  MoveL 5258 to (-75.49, 1.51, -146.03) mm, rotated rx -9.61 ry -16.54 rz -54.03 deg; joints [-10.747, -61.627, 111.301, 199.132, 34.736, -117.948, -415]
  MoveL 5259 to (-75.17, 1.21, -145.97) mm, rotated rx -9.61 ry -16.54 rz -54.03 deg; joints [-10.746, -61.652, 111.337, 199.128, 34.747, -117.942, -415]
  MoveL 5260 to (-74.81, 0.9, -145.93) mm, rotated rx -9.61 ry -16.54 rz -54.03 deg; joints [-10.747, -61.679, 111.378, 199.12, 34.76, -117.933, -415]
  MoveL 5261 to (-74.43, 0.59, -145.92) mm, rotated rx -9.61 ry -16.54 rz -54.03 deg; joints [-10.748, -61.706, 111.42, 199.111, 34.774, -117.923, -415]
  MoveL 5262 to (-74.01, 0.26, -145.91) mm, rotated rx -9.61 ry -16.54 rz -54.03 deg; joints [-10.75, -61.734, 111.466, 199.099, 34.79, -117.911, -415]
  MoveL 5263 to (-73.59, -0.06, -145.91) mm, rotated rx -9.61 ry -16.54 rz -54.03 deg; joints [-10.753, -61.762, 111.51, 199.087, 34.805, -117.899, -415]
  MoveL 5264 to (-73.18, -0.36, -145.93) mm, rotated rx -9.61 ry -16.54 rz -54.03 deg; joints [-10.756, -61.788, 111.554, 199.075, 34.821, -117.886, -415]
  MoveL 5265 to (-72.78, -0.65, -145.94) mm, rotated rx -9.61 ry -16.54 rz -54.03 deg; joints [-10.758, -61.814, 111.596, 199.062, 34.836, -117.873, -415]
  MoveL 5266 to (-72.42, -0.94, -145.92) mm, rotated rx -9.61 ry -16.54 rz -54.03 deg; joints [-10.76, -61.839, 111.636, 199.054, 34.849, -117.864, -415]
  MoveL 5267 to (-72.07, -1.24, -145.88) mm, rotated rx -9.61 ry -16.54 rz -54.03 deg; joints [-10.76, -61.865, 111.675, 199.047, 34.862, -117.855, -415]
  MoveL 5268 to (-71.66, -1.6, -145.83) mm, rotated rx -9.61 ry -16.54 rz -54.03 deg; joints [-10.76, -61.895, 111.722, 199.039, 34.877, -117.846, -415]
  MoveL 5269 to (-71.13, -2.06, -145.77) mm, rotated rx -9.61 ry -16.54 rz -54.03 deg; joints [-10.761, -61.935, 111.781, 199.028, 34.896, -117.834, -415]
  MoveL 5270 to (-70.63, -2.48, -145.75) mm, rotated rx -9.61 ry -16.54 rz -54.03 deg; joints [-10.763, -61.97, 111.836, 199.016, 34.914, -117.821, -415]
  MoveL 5271 to (-68.56, -4.07, -145.75) mm, rotated rx -9.61 ry -16.54 rz -54.03 deg; joints [-10.775, -62.109, 112.059, 198.957, 34.991, -117.76, -415]
  MoveL 5272 to (-68.07, -4.47, -145.71) mm, rotated rx -9.61 ry -16.54 rz -54.03 deg; joints [-10.776, -62.143, 112.112, 198.946, 35.008, -117.748, -415]
  MoveL 5273 to (-67.65, -4.83, -145.65) mm, rotated rx -9.61 ry -16.54 rz -54.03 deg; joints [-10.776, -62.174, 112.159, 198.939, 35.024, -117.739, -415]
  MoveL 5274 to (-67.49, -4.97, -145.51) mm, rotated rx -9.61 ry -16.54 rz -54.03 deg; joints [-10.771, -62.187, 112.178, 198.944, 35.031, -117.741, -415]
  MoveL 5275 to (-67.59, -4.89, -145.24) mm, rotated rx -9.61 ry -16.54 rz -54.03 deg; joints [-10.76, -62.181, 112.17, 198.964, 35.031, -117.754, -415]
  MoveL 5276 to (-67.93, -4.58, -144.84) mm, rotated rx -9.61 ry -16.54 rz -54.03 deg; joints [-10.741, -62.158, 112.136, 198.999, 35.025, -117.78, -415]
  MoveL 5277 to (-68.27, -5.55, -144.03) mm, rotated rx -9.61 ry -16.54 rz -54.03 deg; joints [-10.709, -62.222, 112.153, 199.074, 34.987, -117.841, -415]
  MoveL 5278 to (-67.69, -7.45, -143.82) mm, rotated rx -9.61 ry -16.54 rz -54.03 deg; joints [-10.707, -62.359, 112.27, 199.087, 34.969, -117.855, -415]
  MoveL 5279 to (-67.08, -9.36, -143.66) mm, rotated rx -9.61 ry -16.54 rz -54.03 deg; joints [-10.707, -62.497, 112.39, 199.095, 34.951, -117.865, -415]
  MoveL 5280 to (-66.45, -11.32, -143.5) mm, rotated rx -9.61 ry -16.54 rz -54.03 deg; joints [-10.708, -62.639, 112.512, 199.103, 34.933, -117.875, -415]
  MoveL 5281 to (-65.89, -13.11, -143.21) mm, rotated rx -9.61 ry -16.54 rz -54.03 deg; joints [-10.702, -62.769, 112.625, 199.121, 34.917, -117.892, -415]
  MoveL 5282 to (-65.24, -15.12, -143.02) mm, rotated rx -9.61 ry -16.54 rz -54.03 deg; joints [-10.701, -62.915, 112.75, 199.131, 34.898, -117.904, -415]
  MoveL 5283 to (-64.56, -17.23, -142.84) mm, rotated rx -9.61 ry -16.54 rz -54.03 deg; joints [-10.701, -63.068, 112.882, 199.142, 34.877, -117.917, -415]
  MoveL 5284 to (-63.86, -19.36, -142.75) mm, rotated rx -9.61 ry -16.54 rz -54.03 deg; joints [-10.705, -63.223, 113.014, 199.145, 34.856, -117.925, -415]
  MoveL 5285 to (-63, -21.95, -142.66) mm, rotated rx -9.61 ry -16.54 rz -54.03 deg; joints [-10.711, -63.411, 113.175, 199.149, 34.829, -117.934, -415]
  MoveL 5286 to (-62.38, -23.8, -142.56) mm, rotated rx -9.61 ry -16.54 rz -54.03 deg; joints [-10.713, -63.546, 113.292, 199.153, 34.811, -117.942, -415]
  MoveL 5287 to (-61.8, -25.54, -142.34) mm, rotated rx -9.61 ry -16.54 rz -54.03 deg; joints [-10.711, -63.673, 113.401, 199.166, 34.795, -117.955, -415]
  MoveL 5288 to (-61.16, -27.45, -142.15) mm, rotated rx -9.61 ry -16.54 rz -54.03 deg; joints [-10.71, -63.813, 113.521, 199.177, 34.776, -117.968, -415]
  MoveL 5289 to (-60.47, -29.47, -142.03) mm, rotated rx -9.61 ry -16.54 rz -54.03 deg; joints [-10.712, -63.96, 113.647, 199.183, 34.755, -117.978, -415]
  MoveL 5290 to (-59.79, -31.47, -141.85) mm, rotated rx -9.61 ry -16.54 rz -54.03 deg; joints [-10.712, -64.106, 113.772, 199.193, 34.736, -117.99, -415]
  MoveL 5291 to (-59.11, -33.47, -141.73) mm, rotated rx -9.61 ry -16.54 rz -54.03 deg; joints [-10.715, -64.253, 113.897, 199.2, 34.715, -118, -415]
  MoveL 5292 to (-58.4, -35.53, -141.55) mm, rotated rx -9.61 ry -16.54 rz -54.03 deg; joints [-10.715, -64.404, 114.026, 199.21, 34.694, -118.012, -415]
  MoveL 5293 to (-57.7, -37.55, -141.43) mm, rotated rx -9.61 ry -16.54 rz -54.03 deg; joints [-10.717, -64.551, 114.152, 199.216, 34.673, -118.022, -415]
  MoveL 5294 to (-56.99, -39.56, -141.2) mm, rotated rx -9.61 ry -16.54 rz -54.03 deg; joints [-10.715, -64.7, 114.279, 199.23, 34.653, -118.036, -415]
  MoveL 5295 to (-56.29, -41.58, -141.09) mm, rotated rx -9.61 ry -16.54 rz -54.03 deg; joints [-10.718, -64.848, 114.405, 199.236, 34.631, -118.047, -415]
  MoveL 5296 to (-55.59, -43.59, -140.97) mm, rotated rx -9.61 ry -16.54 rz -54.03 deg; joints [-10.721, -64.996, 114.53, 199.242, 34.609, -118.057, -415]
  MoveL 5297 to (-54.86, -45.6, -140.75) mm, rotated rx -9.61 ry -16.54 rz -54.03 deg; joints [-10.719, -65.144, 114.657, 199.255, 34.59, -118.071, -415]
  MoveL 5298 to (-54.16, -47.41, -140.55) mm, rotated rx -9.61 ry -16.54 rz -54.03 deg; joints [-10.717, -65.279, 114.776, 199.265, 34.575, -118.082, -415]
  MoveL 5299 to (-53.46, -49.03, -140.26) mm, rotated rx -9.61 ry -16.54 rz -54.03 deg; joints [-10.712, -65.401, 114.888, 199.28, 34.567, -118.094, -415]
  MoveL 5300 to (-52.73, -50.49, -139.85) mm, rotated rx -9.61 ry -16.54 rz -54.03 deg; joints [-10.701, -65.514, 114.997, 199.299, 34.566, -118.107, -415]
  MoveL 5301 to (-52.69, -49, -138.92) mm, rotated rx -9.61 ry -16.54 rz -54.03 deg; joints [-10.658, -65.419, 114.96, 199.342, 34.629, -118.12, -415]
  MoveL 5302 to (-52.62, -49.58, -138.91) mm, rotated rx -9.61 ry -16.54 rz -54.03 deg; joints [-10.659, -65.459, 114.984, 199.347, 34.615, -118.128, -415]
  MoveL 5303 to (-52.59, -50.11, -138.89) mm, rotated rx -9.61 ry -16.54 rz -54.03 deg; joints [-10.66, -65.495, 115.005, 199.354, 34.599, -118.137, -415]
  MoveL 5304 to (-52.61, -50.58, -138.83) mm, rotated rx -9.61 ry -16.54 rz -54.03 deg; joints [-10.658, -65.527, 115.02, 199.365, 34.584, -118.148, -415]
  MoveL 5305 to (-52.65, -51.02, -138.76) mm, rotated rx -9.61 ry -16.54 rz -54.03 deg; joints [-10.656, -65.557, 115.032, 199.376, 34.568, -118.16, -415]
  MoveL 5306 to (-52.73, -51.48, -138.71) mm, rotated rx -9.61 ry -16.54 rz -54.03 deg; joints [-10.655, -65.587, 115.042, 199.388, 34.549, -118.174, -415]
  MoveL 5307 to (-52.83, -51.96, -138.68) mm, rotated rx -9.61 ry -16.54 rz -54.03 deg; joints [-10.654, -65.618, 115.05, 199.4, 34.527, -118.188, -415]
  MoveL 5308 to (-52.96, -52.47, -138.66) mm, rotated rx -9.61 ry -16.54 rz -54.03 deg; joints [-10.654, -65.65, 115.057, 199.412, 34.503, -118.203, -415]
  MoveL 5309 to (-53.1, -52.97, -138.66) mm, rotated rx -9.61 ry -16.54 rz -54.03 deg; joints [-10.655, -65.682, 115.063, 199.424, 34.479, -118.217, -415]
  MoveL 5310 to (-53.21, -53.43, -138.65) mm, rotated rx -9.61 ry -16.54 rz -54.03 deg; joints [-10.655, -65.711, 115.07, 199.435, 34.458, -118.23, -415]
  MoveL 5311 to (-53.3, -53.84, -138.63) mm, rotated rx -9.61 ry -16.54 rz -54.03 deg; joints [-10.655, -65.738, 115.077, 199.445, 34.439, -118.242, -415]
  MoveL 5312 to (-53.41, -54.31, -138.61) mm, rotated rx -9.61 ry -16.54 rz -54.03 deg; joints [-10.655, -65.768, 115.083, 199.456, 34.417, -118.256, -415]
  MoveL 5313 to (-53.55, -54.82, -138.61) mm, rotated rx -9.61 ry -16.54 rz -54.03 deg; joints [-10.656, -65.8, 115.089, 199.467, 34.393, -118.27, -415]
  MoveL 5314 to (-53.7, -55.41, -138.59) mm, rotated rx -9.61 ry -16.54 rz -54.03 deg; joints [-10.656, -65.838, 115.097, 199.482, 34.365, -118.288, -415]
  MoveL 5315 to (-53.86, -56.09, -138.55) mm, rotated rx -9.61 ry -16.54 rz -54.03 deg; joints [-10.655, -65.881, 115.108, 199.5, 34.334, -118.309, -415]
  MoveL 5316 to (-54.01, -56.68, -138.53) mm, rotated rx -9.61 ry -16.54 rz -54.03 deg; joints [-10.655, -65.919, 115.116, 199.514, 34.306, -118.326, -415]
  MoveL 5317 to (-54.16, -57.3, -138.51) mm, rotated rx -9.61 ry -16.54 rz -54.03 deg; joints [-10.655, -65.958, 115.125, 199.529, 34.277, -118.344, -415]
  MoveL 5318 to (-54.31, -57.99, -138.47) mm, rotated rx -9.61 ry -16.54 rz -54.03 deg; joints [-10.654, -66.003, 115.136, 199.547, 34.245, -118.365, -415]
  MoveL 5319 to (-54.46, -58.57, -138.45) mm, rotated rx -9.61 ry -16.54 rz -54.03 deg; joints [-10.654, -66.039, 115.143, 199.561, 34.218, -118.382, -415]
  MoveL 5320 to (-54.6, -59.09, -138.45) mm, rotated rx -9.61 ry -16.54 rz -54.03 deg; joints [-10.655, -66.073, 115.15, 199.573, 34.192, -118.397, -415]
  MoveL 5321 to (-55.01, -60.61, -138.45) mm, rotated rx -9.61 ry -16.54 rz -54.03 deg; joints [-10.657, -66.168, 115.167, 199.608, 34.118, -118.442, -415]
  MoveL 5322 to (-55.46, -61.99, -138.54) mm, rotated rx -9.61 ry -16.54 rz -54.03 deg; joints [-10.662, -66.254, 115.176, 199.638, 34.045, -118.482, -415]
  MoveL 5323 to (-55.97, -63.06, -138.79) mm, rotated rx -9.61 ry -16.54 rz -54.03 deg; joints [-10.673, -66.316, 115.169, 199.654, 33.977, -118.511, -415]
  MoveL 5324 to (-56.54, -63.84, -139.21) mm, rotated rx -9.61 ry -16.54 rz -54.03 deg; joints [-10.691, -66.357, 115.145, 199.656, 33.913, -118.53, -415]
  MoveL 5325 to (-56.84, -64.11, -139.48) mm, rotated rx -9.61 ry -16.54 rz -54.03 deg; joints [-10.702, -66.368, 115.127, 199.652, 33.883, -118.536, -415]
  MoveL 5326 to (-57.16, -64.3, -139.8) mm, rotated rx -9.61 ry -16.54 rz -54.03 deg; joints [-10.715, -66.374, 115.105, 199.645, 33.853, -118.539, -415]
  MoveL 5327 to (-57.85, -64.47, -140.56) mm, rotated rx -9.61 ry -16.54 rz -54.03 deg; joints [-10.745, -66.37, 115.05, 199.62, 33.799, -118.536, -415]
  MoveL 5328 to (-58.6, -64.32, -141.49) mm, rotated rx -9.61 ry -16.54 rz -54.03 deg; joints [-10.781, -66.342, 114.977, 199.582, 33.749, -118.523, -415]
  MoveL 5329 to (-60.27, -63.13, -143.85) mm, rotated rx -9.61 ry -16.54 rz -54.03 deg; joints [-10.871, -66.22, 114.784, 199.465, 33.662, -118.464, -415]
  MoveL 5330 to (-61.69, -61.18, -146.21) mm, rotated rx -9.61 ry -16.54 rz -54.03 deg; joints [-10.961, -66.052, 114.587, 199.329, 33.614, -118.38, -415]
  MoveL 5331 to (-62.35, -58.96, -147.9) mm, rotated rx -9.61 ry -16.54 rz -54.03 deg; joints [-11.024, -65.881, 114.445, 199.208, 33.628, -118.292, -415]
  MoveL 5332 to (-62.4, -57.74, -148.49) mm, rotated rx -9.61 ry -16.54 rz -54.03 deg; joints [-11.045, -65.795, 114.396, 199.154, 33.658, -118.246, -415]
  MoveL 5333 to (-62.26, -56.45, -148.91) mm, rotated rx -9.61 ry -16.54 rz -54.03 deg; joints [-11.06, -65.708, 114.36, 199.103, 33.703, -118.199, -415]
  MoveL 5334 to (-61.41, -53.66, -149.25) mm, rotated rx -9.61 ry -16.54 rz -54.03 deg; joints [-11.071, -65.533, 114.331, 199.014, 33.839, -118.101, -415]
  MoveL 5335 to (-59.8, -49.79, -149.25) mm, rotated rx -9.61 ry -16.54 rz -54.03 deg; joints [-11.068, -65.3, 114.329, 198.907, 34.059, -117.97, -415]
  MoveL 5336 to (-59.6, -49.28, -149.27) mm, rotated rx -9.61 ry -16.54 rz -54.03 deg; joints [-11.068, -65.268, 114.327, 198.893, 34.086, -117.952, -415]
  MoveL 5337 to (-59.43, -48.78, -149.31) mm, rotated rx -9.61 ry -16.54 rz -54.03 deg; joints [-11.069, -65.238, 114.324, 198.878, 34.112, -117.935, -415]
  MoveL 5338 to (-59.26, -48.28, -149.37) mm, rotated rx -9.61 ry -16.54 rz -54.03 deg; joints [-11.071, -65.206, 114.319, 198.861, 34.137, -117.918, -415]
  MoveL 5339 to (-59.12, -47.78, -149.45) mm, rotated rx -9.61 ry -16.54 rz -54.03 deg; joints [-11.074, -65.174, 114.313, 198.845, 34.161, -117.9, -415]
  MoveL 5340 to (-58.98, -47.29, -149.53) mm, rotated rx -9.61 ry -16.54 rz -54.03 deg; joints [-11.076, -65.143, 114.307, 198.828, 34.184, -117.883, -415]
  MoveL 5341 to (-58.82, -46.84, -149.57) mm, rotated rx -9.61 ry -16.54 rz -54.03 deg; joints [-11.078, -65.115, 114.304, 198.815, 34.208, -117.867, -415]
  MoveL 5342 to (-58.64, -46.39, -149.59) mm, rotated rx -9.61 ry -16.54 rz -54.03 deg; joints [-11.078, -65.087, 114.303, 198.802, 34.232, -117.852, -415]
  MoveL 5343 to (-58.44, -45.91, -149.59) mm, rotated rx -9.61 ry -16.54 rz -54.03 deg; joints [-11.077, -65.058, 114.302, 198.789, 34.259, -117.836, -415]
  MoveL 5344 to (-58.22, -45.32, -149.62) mm, rotated rx -9.61 ry -16.54 rz -54.03 deg; joints [-11.078, -65.022, 114.299, 198.772, 34.291, -117.816, -415]
  MoveL 5345 to (-57.99, -44.68, -149.68) mm, rotated rx -9.61 ry -16.54 rz -54.03 deg; joints [-11.08, -64.982, 114.295, 198.752, 34.324, -117.793, -415]
  MoveL 5346 to (-57.8, -44.11, -149.7) mm, rotated rx -9.61 ry -16.54 rz -54.03 deg; joints [-11.08, -64.947, 114.291, 198.737, 34.353, -117.776, -415]
  MoveL 5347 to (-57.66, -43.58, -149.71) mm, rotated rx -9.61 ry -16.54 rz -54.03 deg; joints [-11.08, -64.913, 114.283, 198.725, 34.379, -117.761, -415]
  MoveL 5348 to (-57.56, -43.03, -149.71) mm, rotated rx -9.61 ry -16.54 rz -54.03 deg; joints [-11.079, -64.878, 114.272, 198.716, 34.401, -117.748, -415]
  MoveL 5349 to (-57.59, -42.45, -149.71) mm, rotated rx -9.61 ry -16.54 rz -54.03 deg; joints [-11.077, -64.839, 114.251, 198.71, 34.419, -117.74, -415]
  MoveL 5350 to (-57.68, -41.85, -149.71) mm, rotated rx -9.61 ry -16.54 rz -54.03 deg; joints [-11.076, -64.796, 114.223, 198.706, 34.433, -117.734, -415]
  MoveL 5351 to (-57.8, -43.42, -150.67) mm, rotated rx -9.61 ry -16.54 rz -54.03 deg; joints [-11.119, -64.895, 114.258, 198.663, 34.363, -117.722, -415]
  MoveL 5352 to (-58.26, -42.26, -151.09) mm, rotated rx -9.61 ry -16.54 rz -54.03 deg; joints [-11.132, -64.807, 114.177, 198.638, 34.368, -117.704, -415]
  MoveL 5353 to (-58.69, -40.91, -151.42) mm, rotated rx -9.61 ry -16.54 rz -54.03 deg; joints [-11.141, -64.707, 114.094, 198.617, 34.382, -117.685, -415]
  MoveL 5354 to (-59.1, -39.36, -151.67) mm, rotated rx -9.61 ry -16.54 rz -54.03 deg; joints [-11.145, -64.595, 114.006, 198.597, 34.404, -117.666, -415]
  MoveL 5355 to (-59.54, -37.27, -151.78) mm, rotated rx -9.61 ry -16.54 rz -54.03 deg; joints [-11.143, -64.446, 113.898, 198.583, 34.443, -117.646, -415]
  MoveL 5356 to (-60, -35.19, -152.01) mm, rotated rx -9.61 ry -16.54 rz -54.03 deg; joints [-11.145, -64.298, 113.788, 198.561, 34.479, -117.622, -415]
  MoveL 5357 to (-60.43, -33.1, -152.13) mm, rotated rx -9.61 ry -16.54 rz -54.03 deg; joints [-11.143, -64.15, 113.68, 198.546, 34.517, -117.602, -415]
  MoveL 5358 to (-60.86, -31.01, -152.24) mm, rotated rx -9.61 ry -16.54 rz -54.03 deg; joints [-11.141, -64.002, 113.572, 198.531, 34.556, -117.582, -415]
  MoveL 5359 to (-61.3, -28.93, -152.48) mm, rotated rx -9.61 ry -16.54 rz -54.03 deg; joints [-11.143, -63.853, 113.462, 198.509, 34.592, -117.557, -415]
  MoveL 5360 to (-61.73, -26.84, -152.6) mm, rotated rx -9.61 ry -16.54 rz -54.03 deg; joints [-11.141, -63.705, 113.354, 198.495, 34.63, -117.538, -415]
  MoveL 5361 to (-62.15, -24.75, -152.72) mm, rotated rx -9.61 ry -16.54 rz -54.03 deg; joints [-11.139, -63.557, 113.245, 198.48, 34.667, -117.518, -415]
  MoveL 5362 to (-62.64, -22.34, -152.88) mm, rotated rx -9.61 ry -16.54 rz -54.03 deg; joints [-11.137, -63.387, 113.119, 198.462, 34.71, -117.495, -415]
  MoveL 5363 to (-63.05, -20.28, -153.07) mm, rotated rx -9.61 ry -16.54 rz -54.03 deg; joints [-11.139, -63.241, 113.011, 198.443, 34.746, -117.472, -415]
  MoveL 5364 to (-63.5, -18.01, -153.27) mm, rotated rx -9.61 ry -16.54 rz -54.03 deg; joints [-11.139, -63.081, 112.893, 198.423, 34.785, -117.449, -415]
  MoveL 5365 to (-63.93, -15.79, -153.52) mm, rotated rx -9.61 ry -16.54 rz -54.03 deg; joints [-11.142, -62.924, 112.776, 198.4, 34.823, -117.423, -415]
  MoveL 5366 to (-64.34, -13.7, -153.64) mm, rotated rx -9.61 ry -16.54 rz -54.03 deg; joints [-11.14, -62.776, 112.667, 198.385, 34.86, -117.404, -415]
  MoveL 5367 to (-64.76, -11.61, -153.64) mm, rotated rx -9.61 ry -16.54 rz -54.03 deg; joints [-11.133, -62.629, 112.558, 198.38, 34.897, -117.39, -415]
  MoveL 5368 to (-65.16, -9.54, -153.72) mm, rotated rx -9.61 ry -16.54 rz -54.03 deg; joints [-11.13, -62.484, 112.45, 198.369, 34.933, -117.374, -415]
  MoveL 5369 to (-65.53, -7.51, -153.93) mm, rotated rx -9.61 ry -16.54 rz -54.03 deg; joints [-11.132, -62.341, 112.345, 198.349, 34.968, -117.351, -415]
  MoveL 5370 to (-65.92, -5.25, -154.28) mm, rotated rx -9.61 ry -16.54 rz -54.03 deg; joints [-11.139, -62.181, 112.226, 198.318, 35.006, -117.321, -415]
  MoveL 5371 to (-66.23, -3.47, -154.5) mm, rotated rx -9.61 ry -16.54 rz -54.03 deg; joints [-11.142, -62.056, 112.134, 198.299, 35.037, -117.3, -415]
  MoveL 5372 to (-66.63, -1.04, -154.79) mm, rotated rx -9.61 ry -16.54 rz -54.03 deg; joints [-11.146, -61.886, 112.01, 198.271, 35.079, -117.27, -415]
  MoveL 5373 to (-67.03, 1.13, -154.9) mm, rotated rx -9.61 ry -16.54 rz -54.03 deg; joints [-11.144, -61.734, 111.896, 198.258, 35.116, -117.252, -415]
  MoveL 5374 to (-67.44, 3.22, -154.91) mm, rotated rx -9.61 ry -16.54 rz -54.03 deg; joints [-11.137, -61.588, 111.785, 198.253, 35.151, -117.239, -415]
  MoveL 5375 to (-67.1, 4.04, -155.7) mm, rotated rx -9.61 ry -16.54 rz -54.03 deg; joints [-11.169, -61.534, 111.773, 198.182, 35.185, -117.183, -415]
  MoveL 5376 to (-66.85, 3.68, -156.09) mm, rotated rx -9.61 ry -16.54 rz -54.03 deg; joints [-11.187, -61.56, 111.803, 198.152, 35.185, -117.162, -415]
  MoveL 5377 to (-66.78, 3.55, -156.34) mm, rotated rx -9.61 ry -16.54 rz -54.03 deg; joints [-11.198, -61.567, 111.81, 198.134, 35.183, -117.151, -415]
  MoveL 5378 to (-66.88, 3.66, -156.46) mm, rotated rx -9.61 ry -16.54 rz -54.03 deg; joints [-11.202, -61.558, 111.797, 198.129, 35.178, -117.149, -415]
  MoveL 5379 to (-67.14, 3.95, -156.48) mm, rotated rx -9.61 ry -16.54 rz -54.03 deg; joints [-11.201, -61.535, 111.765, 198.134, 35.17, -117.154, -415]
  MoveL 5380 to (-67.47, 4.28, -156.49) mm, rotated rx -9.61 ry -16.54 rz -54.03 deg; joints [-11.199, -61.507, 111.727, 198.142, 35.16, -117.162, -415]
  MoveL 5381 to (-68.58, 5.39, -156.49) mm, rotated rx -9.61 ry -16.54 rz -54.03 deg; joints [-11.192, -61.416, 111.597, 198.171, 35.125, -117.191, -415]
  MoveL 5382 to (-68.96, 5.79, -156.51) mm, rotated rx -9.61 ry -16.54 rz -54.03 deg; joints [-11.19, -61.384, 111.552, 198.18, 35.113, -117.199, -415]
  MoveL 5383 to (-69.33, 6.21, -156.56) mm, rotated rx -9.61 ry -16.54 rz -54.03 deg; joints [-11.189, -61.35, 111.507, 198.186, 35.102, -117.206, -415]
  MoveL 5384 to (-69.7, 6.65, -156.64) mm, rotated rx -9.61 ry -16.54 rz -54.03 deg; joints [-11.19, -61.315, 111.461, 198.19, 35.092, -117.211, -415]
  MoveL 5385 to (-70.06, 7.06, -156.7) mm, rotated rx -9.61 ry -16.54 rz -54.03 deg; joints [-11.19, -61.281, 111.416, 198.195, 35.081, -117.218, -415]
  MoveL 5386 to (-70.42, 7.45, -156.72) mm, rotated rx -9.61 ry -16.54 rz -54.03 deg; joints [-11.189, -61.25, 111.372, 198.202, 35.07, -117.226, -415]
  MoveL 5387 to (-70.76, 7.81, -156.74) mm, rotated rx -9.61 ry -16.54 rz -54.03 deg; joints [-11.187, -61.22, 111.331, 198.21, 35.059, -117.234, -415]
  MoveL 5388 to (-71.06, 8.16, -156.79) mm, rotated rx -9.61 ry -16.54 rz -54.03 deg; joints [-11.187, -61.192, 111.294, 198.215, 35.05, -117.239, -415]
  MoveL 5389 to (-71.36, 8.49, -156.83) mm, rotated rx -9.61 ry -16.54 rz -54.03 deg; joints [-11.186, -61.166, 111.258, 198.219, 35.042, -117.244, -415]
  MoveL 5390 to (-71.7, 8.85, -156.84) mm, rotated rx -9.61 ry -16.54 rz -54.03 deg; joints [-11.185, -61.136, 111.217, 198.227, 35.031, -117.253, -415]
  MoveL 5391 to (-72.1, 9.27, -156.86) mm, rotated rx -9.61 ry -16.54 rz -54.03 deg; joints [-11.183, -61.102, 111.169, 198.237, 35.018, -117.262, -415]
  MoveL 5392 to (-72.57, 9.8, -156.91) mm, rotated rx -9.61 ry -16.54 rz -54.03 deg; joints [-11.182, -61.059, 111.112, 198.245, 35.004, -117.271, -415]
  MoveL 5393 to (-72.98, 10.24, -156.94) mm, rotated rx -9.61 ry -16.54 rz -54.03 deg; joints [-11.18, -61.023, 111.062, 198.254, 34.992, -117.281, -415]
  MoveL 5394 to (-74.47, 11.73, -156.95) mm, rotated rx -9.61 ry -16.54 rz -54.03 deg; joints [-11.171, -60.902, 110.888, 198.293, 34.944, -117.319, -415]
  MoveL 5395 to (-76.32, 13.98, -157.27) mm, rotated rx -9.61 ry -16.54 rz -54.03 deg; joints [-11.171, -60.721, 110.652, 198.317, 34.891, -117.349, -415]
  MoveL 5396 to (-76.94, 15.12, -157.69) mm, rotated rx -9.61 ry -16.54 rz -54.03 deg; joints [-11.182, -60.634, 110.555, 198.303, 34.88, -117.343, -415]
  MoveL 5397 to (-77.36, 16.25, -158.26) mm, rotated rx -9.61 ry -16.54 rz -54.03 deg; joints [-11.201, -60.549, 110.472, 198.271, 34.878, -117.321, -415]
  MoveL 5398 to (-77.61, 18.55, -159.91) mm, rotated rx -9.61 ry -16.54 rz -54.03 deg; joints [-11.261, -60.383, 110.347, 198.155, 34.905, -117.235, -415]
  MoveL 5399 to (-77.06, 20.86, -162.22) mm, rotated rx -9.61 ry -16.54 rz -54.03 deg; joints [-11.35, -60.224, 110.277, 197.969, 34.971, -117.092, -415]
  MoveL 5400 to (-75.98, 22.58, -164.53) mm, rotated rx -9.61 ry -16.54 rz -54.03 deg; joints [-11.443, -60.112, 110.27, 197.77, 35.053, -116.936, -415]
  MoveL 5401 to (-75.35, 22.98, -165.43) mm, rotated rx -9.61 ry -16.54 rz -54.03 deg; joints [-11.482, -60.089, 110.295, 197.687, 35.091, -116.871, -415]
  MoveL 5402 to (-74.66, 23.09, -166.17) mm, rotated rx -9.61 ry -16.54 rz -54.03 deg; joints [-11.514, -60.089, 110.337, 197.615, 35.126, -116.813, -415]
  MoveL 5403 to (-74.29, 23.02, -166.48) mm, rotated rx -9.61 ry -16.54 rz -54.03 deg; joints [-11.528, -60.096, 110.365, 197.583, 35.143, -116.788, -415]
  MoveL 5404 to (-73.91, 22.89, -166.75) mm, rotated rx -9.61 ry -16.54 rz -54.03 deg; joints [-11.541, -60.11, 110.398, 197.554, 35.159, -116.764, -415]
  MoveL 5405 to (-73.09, 22.39, -167.16) mm, rotated rx -9.61 ry -16.54 rz -54.03 deg; joints [-11.562, -60.153, 110.478, 197.503, 35.189, -116.722, -415]
  MoveL 5406 to (-72.21, 21.58, -167.41) mm, rotated rx -9.61 ry -16.54 rz -54.03 deg; joints [-11.578, -60.218, 110.576, 197.463, 35.218, -116.688, -415]
  MoveL 5407 to (-71.28, 20.48, -167.49) mm, rotated rx -9.61 ry -16.54 rz -54.03 deg; joints [-11.589, -60.305, 110.692, 197.434, 35.243, -116.662, -415]
  MoveL 5408 to (-69.04, 17.57, -167.49) mm, rotated rx -9.61 ry -16.54 rz -54.03 deg; joints [-11.606, -60.531, 110.98, 197.38, 35.299, -116.612, -415]
  MoveL 5409 to (-68.76, 17.2, -167.48) mm, rotated rx -9.61 ry -16.54 rz -54.03 deg; joints [-11.607, -60.56, 111.017, 197.374, 35.306, -116.607, -415]
  MoveL 5410 to (-68.53, 16.87, -167.45) mm, rotated rx -9.61 ry -16.54 rz -54.03 deg; joints [-11.608, -60.586, 111.048, 197.371, 35.311, -116.603, -415]
  MoveL 5411 to (-68.25, 16.48, -167.43) mm, rotated rx -9.61 ry -16.54 rz -54.03 deg; joints [-11.61, -60.616, 111.085, 197.365, 35.318, -116.597, -415]
  MoveL 5412 to (-66.01, 13.58, -167.43) mm, rotated rx -9.61 ry -16.54 rz -54.03 deg; joints [-11.627, -60.843, 111.373, 197.311, 35.373, -116.548, -415]
  MoveL 5413 to (-65.69, 13.14, -167.41) mm, rotated rx -9.61 ry -16.54 rz -54.03 deg; joints [-11.629, -60.877, 111.415, 197.305, 35.379, -116.542, -415]
  MoveL 5414 to (-65.4, 12.68, -167.38) mm, rotated rx -9.61 ry -16.54 rz -54.03 deg; joints [-11.63, -60.912, 111.456, 197.301, 35.385, -116.538, -415]
  MoveL 5415 to (-65.19, 12.24, -167.33) mm, rotated rx -9.61 ry -16.54 rz -54.03 deg; joints [-11.63, -60.945, 111.49, 197.3, 35.386, -116.537, -415]
  MoveL 5416 to (-65.05, 11.88, -167.27) mm, rotated rx -9.61 ry -16.54 rz -54.03 deg; joints [-11.629, -60.972, 111.515, 197.302, 35.385, -116.539, -415]
  MoveL 5417 to (-65.01, 11.69, -167.1) mm, rotated rx -9.61 ry -16.54 rz -54.03 deg; joints [-11.623, -60.986, 111.527, 197.313, 35.384, -116.546, -415]
  MoveL 5418 to (-65.04, 11.67, -166.77) mm, rotated rx -9.61 ry -16.54 rz -54.03 deg; joints [-11.61, -60.989, 111.53, 197.335, 35.386, -116.561, -415]
  MoveL 5419 to (-65.12, 11.8, -166.26) mm, rotated rx -9.61 ry -16.54 rz -54.03 deg; joints [-11.588, -60.982, 111.524, 197.37, 35.391, -116.583, -415]
  MoveL 5420 to (-65.63, 11.15, -164.8) mm, rotated rx -9.61 ry -16.54 rz -54.03 deg; joints [-11.528, -61.027, 111.524, 197.486, 35.36, -116.669, -415]
  MoveL 5421 to (-65.35, 6.89, -164.8) mm, rotated rx -9.61 ry -16.54 rz -54.03 deg; joints [-11.541, -61.316, 111.708, 197.51, 35.258, -116.71, -415]
  MoveL 5422 to (-65.22, 4.86, -164.75) mm, rotated rx -9.61 ry -16.54 rz -54.03 deg; joints [-11.545, -61.455, 111.796, 197.525, 35.208, -116.732, -415]
  MoveL 5423 to (-65.1, 2.88, -164.67) mm, rotated rx -9.61 ry -16.54 rz -54.03 deg; joints [-11.547, -61.589, 111.881, 197.542, 35.161, -116.756, -415]
  MoveL 5424 to (-64.97, 0.87, -164.58) mm, rotated rx -9.61 ry -16.54 rz -54.03 deg; joints [-11.55, -61.726, 111.968, 197.56, 35.112, -116.78, -415]
  MoveL 5425 to (-64.84, -1.09, -164.48) mm, rotated rx -9.61 ry -16.54 rz -54.03 deg; joints [-11.551, -61.86, 112.052, 197.579, 35.064, -116.804, -415]
  MoveL 5426 to (-64.73, -3.19, -164.44) mm, rotated rx -9.61 ry -16.54 rz -54.03 deg; joints [-11.556, -62.003, 112.139, 197.595, 35.011, -116.828, -415]
  MoveL 5427 to (-64.69, -5.39, -164.41) mm, rotated rx -9.61 ry -16.54 rz -54.03 deg; joints [-11.561, -62.151, 112.224, 197.615, 34.95, -116.856, -415]
  MoveL 5428 to (-64.43, -7.87, -164.24) mm, rotated rx -9.61 ry -16.54 rz -54.03 deg; joints [-11.562, -62.322, 112.338, 197.638, 34.894, -116.886, -415]
  MoveL 5429 to (-64.28, -10.11, -163.99) mm, rotated rx -9.61 ry -16.54 rz -54.03 deg; joints [-11.558, -62.476, 112.434, 197.669, 34.841, -116.92, -415]
  MoveL 5430 to (-64.14, -12.3, -163.86) mm, rotated rx -9.61 ry -16.54 rz -54.03 deg; joints [-11.559, -62.626, 112.527, 197.692, 34.786, -116.949, -415]
  MoveL 5431 to (-63.99, -14.43, -163.62) mm, rotated rx -9.61 ry -16.54 rz -54.03 deg; joints [-11.556, -62.772, 112.619, 197.722, 34.734, -116.982, -415]
  MoveL 5432 to (-63.84, -16.56, -163.5) mm, rotated rx -9.61 ry -16.54 rz -54.03 deg; joints [-11.557, -62.918, 112.708, 197.744, 34.681, -117.011, -415]
  MoveL 5433 to (-63.69, -18.69, -163.38) mm, rotated rx -9.61 ry -16.54 rz -54.03 deg; joints [-11.559, -63.064, 112.798, 197.766, 34.627, -117.039, -415]
  MoveL 5434 to (-63.53, -20.82, -163.14) mm, rotated rx -9.61 ry -16.54 rz -54.03 deg; joints [-11.555, -63.211, 112.89, 197.796, 34.575, -117.072, -415]
  MoveL 5435 to (-63.37, -22.94, -163.02) mm, rotated rx -9.61 ry -16.54 rz -54.03 deg; joints [-11.557, -63.357, 112.98, 197.819, 34.521, -117.101, -415]
  MoveL 5436 to (-63.21, -25.07, -162.9) mm, rotated rx -9.61 ry -16.54 rz -54.03 deg; joints [-11.558, -63.503, 113.069, 197.841, 34.467, -117.13, -415]
  MoveL 5437 to (-63.05, -27.2, -162.79) mm, rotated rx -9.61 ry -16.54 rz -54.03 deg; joints [-11.56, -63.649, 113.158, 197.864, 34.413, -117.159, -415]
  MoveL 5438 to (-62.86, -29.32, -162.56) mm, rotated rx -9.61 ry -16.54 rz -54.03 deg; joints [-11.557, -63.796, 113.25, 197.893, 34.361, -117.192, -415]
  MoveL 5439 to (-62.7, -31.45, -162.45) mm, rotated rx -9.61 ry -16.54 rz -54.03 deg; joints [-11.559, -63.942, 113.339, 197.916, 34.306, -117.221, -415]
  MoveL 5440 to (-62.51, -33.23, -162.19) mm, rotated rx -9.61 ry -16.54 rz -54.03 deg; joints [-11.554, -64.066, 113.418, 197.944, 34.264, -117.251, -415]
  MoveL 5441 to (-62.33, -34.87, -161.87) mm, rotated rx -9.61 ry -16.54 rz -54.03 deg; joints [-11.546, -64.181, 113.493, 197.976, 34.228, -117.282, -415]
  MoveL 5442 to (-62.12, -36.43, -161.45) mm, rotated rx -9.61 ry -16.54 rz -54.03 deg; joints [-11.534, -64.291, 113.568, 198.013, 34.196, -117.315, -415]
  MoveL 5443 to (-61.52, -34.8, -160.5) mm, rotated rx -9.61 ry -16.54 rz -54.03 deg; joints [-11.492, -64.197, 113.569, 198.039, 34.295, -117.309, -415]
  MoveL 5444 to (-61.52, -35.43, -160.37) mm, rotated rx -9.61 ry -16.54 rz -54.03 deg; joints [-11.488, -64.241, 113.592, 198.054, 34.277, -117.324, -415]
  MoveL 5445 to (-61.58, -36.01, -160.28) mm, rotated rx -9.61 ry -16.54 rz -54.03 deg; joints [-11.486, -64.279, 113.608, 198.068, 34.256, -117.339, -415]
  MoveL 5446 to (-61.75, -36.53, -160.25) mm, rotated rx -9.61 ry -16.54 rz -54.03 deg; joints [-11.485, -64.311, 113.613, 198.082, 34.23, -117.355, -415]
  MoveL 5447 to (-61.96, -37.02, -160.23) mm, rotated rx -9.61 ry -16.54 rz -54.03 deg; joints [-11.485, -64.341, 113.613, 198.096, 34.202, -117.371, -415]
  MoveL 5448 to (-63.78, -40.22, -160.22) mm, rotated rx -9.61 ry -16.54 rz -54.03 deg; joints [-11.486, -64.526, 113.58, 198.195, 33.995, -117.492, -415]
  MoveL 5449 to (-64, -40.62, -160.21) mm, rotated rx -9.61 ry -16.54 rz -54.03 deg; joints [-11.485, -64.55, 113.576, 198.209, 33.969, -117.507, -415]
  MoveL 5450 to (-64.2, -41, -160.18) mm, rotated rx -9.61 ry -16.54 rz -54.03 deg; joints [-11.484, -64.572, 113.574, 198.222, 33.946, -117.522, -415]
  MoveL 5451 to (-64.43, -41.42, -160.17) mm, rotated rx -9.61 ry -16.54 rz -54.03 deg; joints [-11.484, -64.596, 113.57, 198.235, 33.919, -117.538, -415]
  MoveL 5452 to (-64.69, -41.87, -160.17) mm, rotated rx -9.61 ry -16.54 rz -54.03 deg; joints [-11.484, -64.622, 113.565, 198.25, 33.889, -117.556, -415]
  MoveL 5453 to (-65.48, -43.23, -160.17) mm, rotated rx -9.61 ry -16.54 rz -54.03 deg; joints [-11.484, -64.701, 113.549, 198.293, 33.8, -117.608, -415]
  MoveL 5454 to (-65.78, -43.78, -160.15) mm, rotated rx -9.61 ry -16.54 rz -54.03 deg; joints [-11.484, -64.732, 113.544, 198.312, 33.765, -117.63, -415]
  MoveL 5455 to (-66.11, -44.42, -160.12) mm, rotated rx -9.61 ry -16.54 rz -54.03 deg; joints [-11.482, -64.77, 113.54, 198.333, 33.726, -117.655, -415]
  MoveL 5456 to (-66.42, -44.98, -160.09) mm, rotated rx -9.61 ry -16.54 rz -54.03 deg; joints [-11.482, -64.802, 113.535, 198.352, 33.69, -117.677, -415]
  MoveL 5457 to (-66.94, -45.89, -160.09) mm, rotated rx -9.61 ry -16.54 rz -54.03 deg; joints [-11.482, -64.854, 113.524, 198.382, 33.631, -117.713, -415]
  MoveL 5458 to (-67.73, -47.11, -160.18) mm, rotated rx -9.61 ry -16.54 rz -54.03 deg; joints [-11.485, -64.922, 113.502, 198.418, 33.545, -117.76, -415]
  MoveL 5459 to (-68.49, -48.02, -160.43) mm, rotated rx -9.61 ry -16.54 rz -54.03 deg; joints [-11.495, -64.968, 113.47, 198.44, 33.468, -117.794, -415]
  MoveL 5460 to (-69.23, -48.61, -160.85) mm, rotated rx -9.61 ry -16.54 rz -54.03 deg; joints [-11.511, -64.993, 113.426, 198.445, 33.4, -117.815, -415]
  MoveL 5461 to (-69.6, -48.79, -161.12) mm, rotated rx -9.61 ry -16.54 rz -54.03 deg; joints [-11.521, -64.997, 113.401, 198.442, 33.37, -117.82, -415]
  MoveL 5462 to (-69.96, -48.9, -161.44) mm, rotated rx -9.61 ry -16.54 rz -54.03 deg; joints [-11.533, -64.996, 113.372, 198.435, 33.341, -117.822, -415]
  MoveL 5463 to (-70.66, -48.87, -162.19) mm, rotated rx -9.61 ry -16.54 rz -54.03 deg; joints [-11.562, -64.977, 113.308, 198.408, 33.292, -117.816, -415]
  MoveL 5464 to (-71.34, -48.53, -163.12) mm, rotated rx -9.61 ry -16.54 rz -54.03 deg; joints [-11.596, -64.937, 113.232, 198.366, 33.251, -117.796, -415]
  MoveL 5465 to (-72.65, -46.92, -165.47) mm, rotated rx -9.61 ry -16.54 rz -54.03 deg; joints [-11.684, -64.792, 113.049, 198.234, 33.197, -117.717, -415]
  MoveL 5466 to (-73.51, -44.65, -167.82) mm, rotated rx -9.61 ry -16.54 rz -54.03 deg; joints [-11.771, -64.611, 112.879, 198.079, 33.188, -117.61, -415]
  MoveL 5467 to (-73.58, -42.31, -169.5) mm, rotated rx -9.61 ry -16.54 rz -54.03 deg; joints [-11.834, -64.443, 112.776, 197.941, 33.237, -117.501, -415]
  MoveL 5468 to (-73.31, -41.11, -170.09) mm, rotated rx -9.61 ry -16.54 rz -54.03 deg; joints [-11.856, -64.364, 112.75, 197.878, 33.283, -117.445, -415]
  MoveL 5469 to (-72.85, -39.89, -170.51) mm, rotated rx -9.61 ry -16.54 rz -54.03 deg; joints [-11.872, -64.288, 112.741, 197.82, 33.343, -117.39, -415]
  MoveL 5470 to (-71.32, -37.41, -170.85) mm, rotated rx -9.61 ry -16.54 rz -54.03 deg; joints [-11.886, -64.146, 112.773, 197.716, 33.507, -117.277, -415]
  MoveL 5471 to (-69.41, -34.91, -170.85) mm, rotated rx -9.61 ry -16.54 rz -54.03 deg; joints [-11.888, -64.011, 112.838, 197.622, 33.697, -117.166, -415]
  MoveL 5472 to (-68.85, -34.1, -170.89) mm, rotated rx -9.61 ry -16.54 rz -54.03 deg; joints [-11.89, -63.966, 112.854, 197.591, 33.755, -117.131, -415]
  MoveL 5473 to (-68.53, -33.69, -170.89) mm, rotated rx -9.61 ry -16.54 rz -54.03 deg; joints [-11.89, -63.944, 112.864, 197.575, 33.786, -117.112, -415]
  MoveL 5474 to (-68.21, -33.26, -170.9) mm, rotated rx -9.61 ry -16.54 rz -54.03 deg; joints [-11.89, -63.92, 112.875, 197.559, 33.819, -117.093, -415]
  MoveL 5475 to (-67.87, -32.8, -170.92) mm, rotated rx -9.61 ry -16.54 rz -54.03 deg; joints [-11.892, -63.895, 112.885, 197.541, 33.852, -117.073, -415]
  MoveL 5476 to (-67.51, -32.26, -170.98) mm, rotated rx -9.61 ry -16.54 rz -54.03 deg; joints [-11.894, -63.865, 112.895, 197.519, 33.89, -117.048, -415]
  MoveL 5477 to (-67.18, -31.79, -171.01) mm, rotated rx -9.61 ry -16.54 rz -54.03 deg; joints [-11.896, -63.838, 112.905, 197.501, 33.924, -117.027, -415]
  MoveL 5478 to (-66.87, -31.36, -171.02) mm, rotated rx -9.61 ry -16.54 rz -54.03 deg; joints [-11.896, -63.815, 112.914, 197.485, 33.955, -117.009, -415]
  MoveL 5479 to (-66.59, -30.97, -171.05) mm, rotated rx -9.61 ry -16.54 rz -54.03 deg; joints [-11.898, -63.793, 112.922, 197.469, 33.983, -116.991, -415]
  MoveL 5480 to (-66.35, -30.59, -171.1) mm, rotated rx -9.61 ry -16.54 rz -54.03 deg; joints [-11.9, -63.771, 112.927, 197.453, 34.009, -116.974, -415]
  MoveL 5481 to (-66.09, -30.21, -171.14) mm, rotated rx -9.61 ry -16.54 rz -54.03 deg; joints [-11.901, -63.75, 112.934, 197.438, 34.035, -116.958, -415]
  MoveL 5482 to (-65.79, -29.8, -171.15) mm, rotated rx -9.61 ry -16.54 rz -54.03 deg; joints [-11.902, -63.727, 112.943, 197.423, 34.066, -116.94, -415]
  MoveL 5483 to (-65.49, -29.38, -171.16) mm, rotated rx -9.61 ry -16.54 rz -54.03 deg; joints [-11.902, -63.704, 112.952, 197.408, 34.096, -116.922, -415]
  MoveL 5484 to (-65.2, -28.95, -171.17) mm, rotated rx -9.61 ry -16.54 rz -54.03 deg; joints [-11.903, -63.68, 112.959, 197.394, 34.126, -116.905, -415]
  MoveL 5485 to (-64.98, -28.52, -171.18) mm, rotated rx -9.61 ry -16.54 rz -54.03 deg; joints [-11.903, -63.654, 112.961, 197.38, 34.153, -116.889, -415]
  MoveL 5486 to (-64.82, -28.07, -171.22) mm, rotated rx -9.61 ry -16.54 rz -54.03 deg; joints [-11.904, -63.626, 112.958, 197.368, 34.176, -116.876, -415]
  MoveL 5487 to (-64.72, -27.63, -171.26) mm, rotated rx -9.61 ry -16.54 rz -54.03 deg; joints [-11.905, -63.598, 112.949, 197.358, 34.194, -116.864, -415]
  MoveL 5488 to (-64.66, -27.17, -171.31) mm, rotated rx -9.61 ry -16.54 rz -54.03 deg; joints [-11.906, -63.568, 112.938, 197.349, 34.212, -116.853, -415]
  MoveL 5489 to (-65.12, -28.63, -172.27) mm, rotated rx -9.61 ry -16.54 rz -54.03 deg; joints [-11.948, -63.652, 112.942, 197.313, 34.127, -116.849, -415]
  MoveL 5490 to (-65.18, -26.91, -172.65) mm, rotated rx -9.61 ry -16.54 rz -54.03 deg; joints [-11.958, -63.533, 112.872, 197.274, 34.172, -116.812, -415]
  MoveL 5491 to (-65.19, -25.1, -172.93) mm, rotated rx -9.61 ry -16.54 rz -54.03 deg; joints [-11.965, -63.41, 112.805, 197.24, 34.224, -116.776, -415]
  MoveL 5492 to (-65.15, -23.15, -173.13) mm, rotated rx -9.61 ry -16.54 rz -54.03 deg; joints [-11.967, -63.279, 112.737, 197.207, 34.283, -116.739, -415]
  MoveL 5493 to (-65.07, -21.02, -173.35) mm, rotated rx -9.61 ry -16.54 rz -54.03 deg; joints [-11.971, -63.136, 112.665, 197.171, 34.35, -116.698, -415]
  MoveL 5494 to (-64.96, -18.89, -173.47) mm, rotated rx -9.61 ry -16.54 rz -54.03 deg; joints [-11.97, -62.995, 112.596, 197.141, 34.42, -116.661, -415]
  MoveL 5495 to (-64.84, -16.75, -173.58) mm, rotated rx -9.61 ry -16.54 rz -54.03 deg; joints [-11.969, -62.853, 112.526, 197.112, 34.49, -116.625, -415]
  MoveL 5496 to (-64.75, -14.62, -173.81) mm, rotated rx -9.61 ry -16.54 rz -54.03 deg; joints [-11.973, -62.71, 112.454, 197.075, 34.557, -116.584, -415]
  MoveL 5497 to (-64.63, -12.49, -173.93) mm, rotated rx -9.61 ry -16.54 rz -54.03 deg; joints [-11.972, -62.568, 112.385, 197.046, 34.626, -116.547, -415]
  MoveL 5498 to (-64.51, -10.36, -174.05) mm, rotated rx -9.61 ry -16.54 rz -54.03 deg; joints [-11.971, -62.427, 112.315, 197.016, 34.695, -116.511, -415]
  MoveL 5499 to (-64.39, -8.22, -174.29) mm, rotated rx -9.61 ry -16.54 rz -54.03 deg; joints [-11.975, -62.284, 112.244, 196.98, 34.762, -116.47, -415]
  MoveL 5500 to (-64.26, -6.09, -174.41) mm, rotated rx -9.61 ry -16.54 rz -54.03 deg; joints [-11.975, -62.143, 112.174, 196.951, 34.83, -116.434, -415]
  MoveL 5501 to (-64.13, -3.96, -174.53) mm, rotated rx -9.61 ry -16.54 rz -54.03 deg; joints [-11.974, -62.001, 112.104, 196.922, 34.899, -116.398, -415]
  MoveL 5502 to (-64.01, -1.95, -174.72) mm, rotated rx -9.61 ry -16.54 rz -54.03 deg; joints [-11.977, -61.867, 112.037, 196.89, 34.963, -116.362, -415]
  MoveL 5503 to (-63.89, -0.13, -174.94) mm, rotated rx -9.61 ry -16.54 rz -54.03 deg; joints [-11.981, -61.745, 111.976, 196.858, 35.02, -116.326, -415]
  MoveL 5504 to (-63.76, 1.83, -175.04) mm, rotated rx -9.61 ry -16.54 rz -54.03 deg; joints [-11.98, -61.616, 111.911, 196.832, 35.082, -116.294, -415]
  MoveL 5505 to (-63.73, 4, -175.04) mm, rotated rx -9.61 ry -16.54 rz -54.03 deg; joints [-11.974, -61.471, 111.832, 196.815, 35.147, -116.268, -415]
  MoveL 5506 to (-63.53, 6.72, -175.13) mm, rotated rx -9.61 ry -16.54 rz -54.03 deg; joints [-11.971, -61.291, 111.744, 196.783, 35.234, -116.225, -415]
  MoveL 5507 to (-63.25, 9.16, -175.37) mm, rotated rx -9.61 ry -16.54 rz -54.03 deg; joints [-11.975, -61.13, 111.67, 196.74, 35.318, -116.177, -415]
  MoveL 5508 to (-63.1, 11.19, -175.55) mm, rotated rx -9.61 ry -16.54 rz -54.03 deg; joints [-11.977, -60.995, 111.602, 196.71, 35.382, -116.142, -415]
  MoveL 5509 to (-62.95, 13.06, -175.87) mm, rotated rx -9.61 ry -16.54 rz -54.03 deg; joints [-11.986, -60.87, 111.539, 196.671, 35.439, -116.102, -415]
  MoveL 5510 to (-62.79, 15.1, -176.05) mm, rotated rx -9.61 ry -16.54 rz -54.03 deg; joints [-11.988, -60.735, 111.471, 196.64, 35.503, -116.067, -415]
  MoveL 5511 to (-62.62, 17.06, -176.25) mm, rotated rx -9.61 ry -16.54 rz -54.03 deg; joints [-11.991, -60.604, 111.406, 196.609, 35.565, -116.031, -415]
  MoveL 5512 to (-62.42, 18.98, -176.54) mm, rotated rx -9.61 ry -16.54 rz -54.03 deg; joints [-11.998, -60.477, 111.344, 196.571, 35.627, -115.992, -415]
  MoveL 5513 to (-61.83, 19.67, -177.3) mm, rotated rx -9.61 ry -16.54 rz -54.03 deg; joints [-12.03, -60.434, 111.355, 196.499, 35.672, -115.933, -415]
  MoveL 5514 to (-61.66, 19.34, -177.68) mm, rotated rx -9.61 ry -16.54 rz -54.03 deg; joints [-12.047, -60.456, 111.376, 196.471, 35.668, -115.915, -415]
  MoveL 5515 to (-61.6, 19.28, -177.93) mm, rotated rx -9.61 ry -16.54 rz -54.03 deg; joints [-12.057, -60.46, 111.38, 196.454, 35.667, -115.904, -415]
  MoveL 5516 to (-61.66, 19.48, -178.05) mm, rotated rx -9.61 ry -16.54 rz -54.03 deg; joints [-12.062, -60.444, 111.367, 196.447, 35.668, -115.899, -415]
  MoveL 5517 to (-61.87, 19.96, -178.1) mm, rotated rx -9.61 ry -16.54 rz -54.03 deg; joints [-12.061, -60.409, 111.331, 196.447, 35.668, -115.899, -415]
  MoveL 5518 to (-62.17, 20.56, -178.14) mm, rotated rx -9.61 ry -16.54 rz -54.03 deg; joints [-12.06, -60.364, 111.284, 196.451, 35.666, -115.902, -415]
  MoveL 5519 to (-62.96, 21.92, -178.14) mm, rotated rx -9.61 ry -16.54 rz -54.03 deg; joints [-12.052, -60.262, 111.169, 196.468, 35.655, -115.916, -415]
  MoveL 5520 to (-63.23, 22.39, -178.15) mm, rotated rx -9.61 ry -16.54 rz -54.03 deg; joints [-12.05, -60.227, 111.129, 196.473, 35.651, -115.921, -415]
  MoveL 5521 to (-63.48, 22.86, -178.17) mm, rotated rx -9.61 ry -16.54 rz -54.03 deg; joints [-12.048, -60.192, 111.091, 196.477, 35.648, -115.924, -415]
  MoveL 5522 to (-63.73, 23.35, -178.22) mm, rotated rx -9.61 ry -16.54 rz -54.03 deg; joints [-12.048, -60.155, 111.051, 196.479, 35.646, -115.926, -415]
  MoveL 5523 to (-63.97, 23.86, -178.29) mm, rotated rx -9.61 ry -16.54 rz -54.03 deg; joints [-12.048, -60.117, 111.012, 196.479, 35.644, -115.926, -415]
  MoveL 5524 to (-64.21, 24.36, -178.35) mm, rotated rx -9.61 ry -16.54 rz -54.03 deg; joints [-12.048, -60.08, 110.973, 196.48, 35.642, -115.927, -415]
  MoveL 5525 to (-64.45, 24.79, -178.37) mm, rotated rx -9.61 ry -16.54 rz -54.03 deg; joints [-12.047, -60.047, 110.937, 196.484, 35.639, -115.93, -415]
  MoveL 5526 to (-64.67, 25.19, -178.39) mm, rotated rx -9.61 ry -16.54 rz -54.03 deg; joints [-12.045, -60.018, 110.904, 196.487, 35.637, -115.933, -415]
  MoveL 5527 to (-65.46, 26.55, -178.39) mm, rotated rx -9.61 ry -16.54 rz -54.03 deg; joints [-12.038, -59.916, 110.789, 196.505, 35.625, -115.948, -415]
  MoveL 5528 to (-65.71, 27.01, -178.4) mm, rotated rx -9.61 ry -16.54 rz -54.03 deg; joints [-12.036, -59.882, 110.751, 196.509, 35.622, -115.952, -415]
  MoveL 5529 to (-65.93, 27.43, -178.43) mm, rotated rx -9.61 ry -16.54 rz -54.03 deg; joints [-12.035, -59.85, 110.716, 196.512, 35.619, -115.954, -415]
  MoveL 5530 to (-66.13, 27.83, -178.48) mm, rotated rx -9.61 ry -16.54 rz -54.03 deg; joints [-12.035, -59.82, 110.685, 196.513, 35.618, -115.955, -415]
  MoveL 5531 to (-66.33, 28.23, -178.52) mm, rotated rx -9.61 ry -16.54 rz -54.03 deg; joints [-12.034, -59.79, 110.652, 196.515, 35.616, -115.957, -415]
  MoveL 5532 to (-66.57, 28.66, -178.53) mm, rotated rx -9.61 ry -16.54 rz -54.03 deg; joints [-12.032, -59.758, 110.617, 196.519, 35.612, -115.96, -415]
  MoveL 5533 to (-66.83, 29.11, -178.53) mm, rotated rx -9.61 ry -16.54 rz -54.03 deg; joints [-12.03, -59.724, 110.578, 196.525, 35.608, -115.965, -415]
  MoveL 5534 to (-68.05, 31.78, -178.87) mm, rotated rx -9.61 ry -16.54 rz -54.03 deg; joints [-12.031, -59.527, 110.373, 196.527, 35.601, -115.968, -415]
  MoveL 5535 to (-68.37, 33.06, -179.29) mm, rotated rx -9.61 ry -16.54 rz -54.03 deg; joints [-12.042, -59.434, 110.292, 196.503, 35.61, -115.95, -415]
  MoveL 5536 to (-68.49, 34.3, -179.88) mm, rotated rx -9.61 ry -16.54 rz -54.03 deg; joints [-12.062, -59.346, 110.226, 196.462, 35.627, -115.919, -415]
  MoveL 5537 to (-68.17, 36.66, -181.57) mm, rotated rx -9.61 ry -16.54 rz -54.03 deg; joints [-12.125, -59.182, 110.137, 196.332, 35.688, -115.818, -415]
  MoveL 5538 to (-67.08, 38.87, -183.93) mm, rotated rx -9.61 ry -16.54 rz -54.03 deg; joints [-12.218, -59.035, 110.106, 196.136, 35.783, -115.666, -415]
  MoveL 5539 to (-65.63, 40.37, -186.3) mm, rotated rx -9.61 ry -16.54 rz -54.03 deg; joints [-12.315, -58.939, 110.13, 195.933, 35.882, -115.509, -415]
  MoveL 5540 to (-64.93, 40.65, -187.23) mm, rotated rx -9.61 ry -16.54 rz -54.03 deg; joints [-12.355, -58.924, 110.162, 195.852, 35.92, -115.446, -415]
  MoveL 5541 to (-64.25, 40.61, -187.98) mm, rotated rx -9.61 ry -16.54 rz -54.03 deg; joints [-12.388, -58.931, 110.208, 195.783, 35.952, -115.394, -415]
  MoveL 5542 to (-63.91, 40.47, -188.3) mm, rotated rx -9.61 ry -16.54 rz -54.03 deg; joints [-12.403, -58.943, 110.236, 195.753, 35.965, -115.371, -415]
  MoveL 5543 to (-63.57, 40.25, -188.58) mm, rotated rx -9.61 ry -16.54 rz -54.03 deg; joints [-12.416, -58.96, 110.268, 195.726, 35.977, -115.351, -415]
  MoveL 5544 to (-62.92, 39.58, -189) mm, rotated rx -9.61 ry -16.54 rz -54.03 deg; joints [-12.438, -59.011, 110.341, 195.682, 35.995, -115.318, -415]
  MoveL 5545 to (-62.28, 38.59, -189.25) mm, rotated rx -9.61 ry -16.54 rz -54.03 deg; joints [-12.454, -59.084, 110.428, 195.651, 36.005, -115.295, -415]
  MoveL 5546 to (-61.65, 37.29, -189.34) mm, rotated rx -9.61 ry -16.54 rz -54.03 deg; joints [-12.465, -59.179, 110.528, 195.633, 36.008, -115.282, -415]
  MoveL 5547 to (-61.04, 35.84, -189.34) mm, rotated rx -9.61 ry -16.54 rz -54.03 deg; joints [-12.472, -59.284, 110.634, 195.621, 36.008, -115.274, -415]
  MoveL 5548 to (-60.84, 35.35, -189.33) mm, rotated rx -9.61 ry -16.54 rz -54.03 deg; joints [-12.474, -59.32, 110.67, 195.617, 36.008, -115.272, -415]
  MoveL 5549 to (-60.64, 34.81, -189.3) mm, rotated rx -9.61 ry -16.54 rz -54.03 deg; joints [-12.476, -59.359, 110.707, 195.616, 36.006, -115.271, -415]
  MoveL 5550 to (-60.43, 34.2, -189.23) mm, rotated rx -9.61 ry -16.54 rz -54.03 deg; joints [-12.476, -59.403, 110.749, 195.616, 36.003, -115.273, -415]
  MoveL 5551 to (-60.23, 33.67, -189.21) mm, rotated rx -9.61 ry -16.54 rz -54.03 deg; joints [-12.477, -59.441, 110.786, 195.614, 36.002, -115.271, -415]
  MoveL 5552 to (-60.03, 33.19, -189.2) mm, rotated rx -9.61 ry -16.54 rz -54.03 deg; joints [-12.48, -59.477, 110.821, 195.61, 36.002, -115.269, -415]
  MoveL 5553 to (-59.83, 32.71, -189.19) mm, rotated rx -9.61 ry -16.54 rz -54.03 deg; joints [-12.482, -59.511, 110.856, 195.607, 36.001, -115.267, -415]
  MoveL 5554 to (-59.66, 32.22, -189.15) mm, rotated rx -9.61 ry -16.54 rz -54.03 deg; joints [-12.482, -59.546, 110.889, 195.607, 35.999, -115.268, -415]
  MoveL 5555 to (-59.52, 31.75, -189.07) mm, rotated rx -9.61 ry -16.54 rz -54.03 deg; joints [-12.481, -59.581, 110.92, 195.61, 35.996, -115.27, -415]
  MoveL 5556 to (-59.38, 31.26, -188.97) mm, rotated rx -9.61 ry -16.54 rz -54.03 deg; joints [-12.479, -59.616, 110.951, 195.615, 35.993, -115.274, -415]
  MoveL 5557 to (-59.23, 30.77, -188.9) mm, rotated rx -9.61 ry -16.54 rz -54.03 deg; joints [-12.479, -59.651, 110.984, 195.617, 35.99, -115.276, -415]
  MoveL 5558 to (-59.04, 30.27, -188.87) mm, rotated rx -9.61 ry -16.54 rz -54.03 deg; joints [-12.48, -59.687, 111.018, 195.615, 35.989, -115.275, -415]
  MoveL 5559 to (-58.85, 29.79, -188.86) mm, rotated rx -9.61 ry -16.54 rz -54.03 deg; joints [-12.482, -59.722, 111.053, 195.612, 35.988, -115.273, -415]
  MoveL 5560 to (-57.89, 27.42, -188.85) mm, rotated rx -9.61 ry -16.54 rz -54.03 deg; joints [-12.493, -59.894, 111.221, 195.595, 35.983, -115.263, -415]
  MoveL 5561 to (-57.8, 27.04, -188.83) mm, rotated rx -9.61 ry -16.54 rz -54.03 deg; joints [-12.494, -59.921, 111.244, 195.595, 35.978, -115.264, -415]
  MoveL 5562 to (-57.78, 26.88, -188.71) mm, rotated rx -9.61 ry -16.54 rz -54.03 deg; joints [-12.49, -59.933, 111.253, 195.603, 35.976, -115.27, -415]
  MoveL 5563 to (-57.8, 26.96, -188.48) mm, rotated rx -9.61 ry -16.54 rz -54.03 deg; joints [-12.48, -59.928, 111.251, 195.618, 35.98, -115.279, -415]
  MoveL 5564 to (-57.86, 27.32, -188.12) mm, rotated rx -9.61 ry -16.54 rz -54.03 deg; joints [-12.464, -59.906, 111.237, 195.641, 35.991, -115.291, -415]
  MoveL 5565 to (-58.39, 26.76, -187.38) mm, rotated rx -9.61 ry -16.54 rz -54.03 deg; joints [-12.433, -59.941, 111.226, 195.707, 35.952, -115.344, -415]
  MoveL 5566 to (-58.8, 24.68, -187.36) mm, rotated rx -9.61 ry -16.54 rz -54.03 deg; joints [-12.437, -60.075, 111.277, 195.732, 35.871, -115.379, -415]
  MoveL 5567 to (-59.24, 22.54, -187.23) mm, rotated rx -9.61 ry -16.54 rz -54.03 deg; joints [-12.436, -60.213, 111.327, 195.767, 35.787, -115.42, -415]
  MoveL 5568 to (-59.74, 20.33, -186.97) mm, rotated rx -9.61 ry -16.54 rz -54.03 deg; joints [-12.43, -60.357, 111.378, 195.812, 35.699, -115.469, -415]
  MoveL 5569 to (-60.18, 18.25, -186.84) mm, rotated rx -9.61 ry -16.54 rz -54.03 deg; joints [-12.429, -60.49, 111.426, 195.846, 35.617, -115.511, -415]
  MoveL 5570 to (-60.61, 16.25, -186.58) mm, rotated rx -9.61 ry -16.54 rz -54.03 deg; joints [-12.422, -60.62, 111.474, 195.888, 35.539, -115.556, -415]
  MoveL 5571 to (-61.06, 14.2, -186.22) mm, rotated rx -9.61 ry -16.54 rz -54.03 deg; joints [-12.412, -60.754, 111.522, 195.938, 35.458, -115.607, -415]
  MoveL 5572 to (-61.49, 12.09, -186.09) mm, rotated rx -9.61 ry -16.54 rz -54.03 deg; joints [-12.411, -60.889, 111.571, 195.973, 35.375, -115.65, -415]
  MoveL 5573 to (-61.9, 10.02, -185.99) mm, rotated rx -9.61 ry -16.54 rz -54.03 deg; joints [-12.411, -61.023, 111.619, 196.006, 35.293, -115.69, -415]
  MoveL 5574 to (-62.32, 7.91, -185.84) mm, rotated rx -9.61 ry -16.54 rz -54.03 deg; joints [-12.409, -61.159, 111.669, 196.042, 35.21, -115.733, -415]
  MoveL 5575 to (-62.75, 5.87, -185.55) mm, rotated rx -9.61 ry -16.54 rz -54.03 deg; joints [-12.402, -61.291, 111.716, 196.088, 35.13, -115.782, -415]
  MoveL 5576 to (-63.13, 3.72, -185.21) mm, rotated rx -9.61 ry -16.54 rz -54.03 deg; joints [-12.393, -61.432, 111.771, 196.137, 35.049, -115.833, -415]
  MoveL 5577 to (-63.53, 1.63, -185.03) mm, rotated rx -9.61 ry -16.54 rz -54.03 deg; joints [-12.39, -61.567, 111.821, 196.175, 34.968, -115.878, -415]
  MoveL 5578 to (-63.92, -0.48, -184.92) mm, rotated rx -9.61 ry -16.54 rz -54.03 deg; joints [-12.39, -61.703, 111.87, 196.21, 34.885, -115.92, -415]
  MoveL 5579 to (-64.32, -2.56, -184.85) mm, rotated rx -9.61 ry -16.54 rz -54.03 deg; joints [-12.392, -61.837, 111.918, 196.242, 34.801, -115.96, -415]
  MoveL 5580 to (-64.7, -4.67, -184.63) mm, rotated rx -9.61 ry -16.54 rz -54.03 deg; joints [-12.387, -61.974, 111.969, 196.284, 34.72, -116.007, -415]
  MoveL 5581 to (-65.08, -6.76, -184.49) mm, rotated rx -9.61 ry -16.54 rz -54.03 deg; joints [-12.386, -62.109, 112.017, 196.321, 34.637, -116.051, -415]
  MoveL 5582 to (-65.48, -8.87, -184.41) mm, rotated rx -9.61 ry -16.54 rz -54.03 deg; joints [-12.387, -62.244, 112.065, 196.354, 34.552, -116.093, -415]
  MoveL 5583 to (-65.84, -10.96, -184.18) mm, rotated rx -9.61 ry -16.54 rz -54.03 deg; joints [-12.383, -62.38, 112.116, 196.397, 34.472, -116.14, -415]
  MoveL 5584 to (-66.19, -13.08, -183.95) mm, rotated rx -9.61 ry -16.54 rz -54.03 deg; joints [-12.378, -62.518, 112.168, 196.44, 34.39, -116.189, -415]
  MoveL 5585 to (-66.57, -15.23, -183.8) mm, rotated rx -9.61 ry -16.54 rz -54.03 deg; joints [-12.377, -62.657, 112.218, 196.48, 34.306, -116.235, -415]
  MoveL 5586 to (-66.86, -17.09, -183.68) mm, rotated rx -9.61 ry -16.54 rz -54.03 deg; joints [-12.376, -62.777, 112.263, 196.512, 34.234, -116.273, -415]
  MoveL 5587 to (-67.06, -18.71, -183.47) mm, rotated rx -9.61 ry -16.54 rz -54.03 deg; joints [-12.371, -62.884, 112.309, 196.545, 34.176, -116.31, -415]
  MoveL 5588 to (-67.16, -20.15, -183.14) mm, rotated rx -9.61 ry -16.54 rz -54.03 deg; joints [-12.362, -62.98, 112.356, 196.582, 34.131, -116.345, -415]
  MoveL 5589 to (-66.66, -18.76, -182.19) mm, rotated rx -9.61 ry -16.54 rz -54.03 deg; joints [-12.321, -62.902, 112.357, 196.618, 34.214, -116.35, -415]
  MoveL 5590 to (-66.75, -19.25, -182.19) mm, rotated rx -9.61 ry -16.54 rz -54.03 deg; joints [-12.322, -62.933, 112.367, 196.625, 34.194, -116.36, -415]
  MoveL 5591 to (-66.89, -19.73, -182.18) mm, rotated rx -9.61 ry -16.54 rz -54.03 deg; joints [-12.322, -62.963, 112.373, 196.634, 34.171, -116.371, -415]
  MoveL 5592 to (-67.12, -20.21, -182.16) mm, rotated rx -9.61 ry -16.54 rz -54.03 deg; joints [-12.322, -62.991, 112.372, 196.647, 34.143, -116.387, -415]
  MoveL 5593 to (-67.42, -20.68, -182.12) mm, rotated rx -9.61 ry -16.54 rz -54.03 deg; joints [-12.32, -63.019, 112.366, 196.664, 34.111, -116.406, -415]
  MoveL 5594 to (-67.79, -21.17, -182.06) mm, rotated rx -9.61 ry -16.54 rz -54.03 deg; joints [-12.317, -63.046, 112.355, 196.685, 34.075, -116.428, -415]
  MoveL 5595 to (-68.18, -21.6, -182.02) mm, rotated rx -9.61 ry -16.54 rz -54.03 deg; joints [-12.315, -63.069, 112.34, 196.704, 34.04, -116.45, -415]
  MoveL 5596 to (-68.57, -22.01, -182.01) mm, rotated rx -9.61 ry -16.54 rz -54.03 deg; joints [-12.314, -63.09, 112.324, 196.722, 34.004, -116.47, -415]
  MoveL 5597 to (-68.94, -22.38, -182.01) mm, rotated rx -9.61 ry -16.54 rz -54.03 deg; joints [-12.313, -63.109, 112.309, 196.738, 33.971, -116.489, -415]
  MoveL 5598 to (-69.3, -22.76, -182) mm, rotated rx -9.61 ry -16.54 rz -54.03 deg; joints [-12.313, -63.128, 112.293, 196.754, 33.938, -116.508, -415]
  MoveL 5599 to (-69.7, -23.2, -181.96) mm, rotated rx -9.61 ry -16.54 rz -54.03 deg; joints [-12.31, -63.151, 112.278, 196.774, 33.902, -116.53, -415]
  MoveL 5600 to (-70.11, -23.71, -181.87) mm, rotated rx -9.61 ry -16.54 rz -54.03 deg; joints [-12.306, -63.179, 112.264, 196.799, 33.863, -116.556, -415]
  MoveL 5601 to (-70.45, -24.1, -181.82) mm, rotated rx -9.61 ry -16.54 rz -54.03 deg; joints [-12.304, -63.2, 112.252, 196.817, 33.831, -116.576, -415]
  MoveL 5602 to (-70.74, -24.41, -181.8) mm, rotated rx -9.61 ry -16.54 rz -54.03 deg; joints [-12.302, -63.216, 112.24, 196.832, 33.805, -116.592, -415]
  MoveL 5603 to (-71.08, -24.76, -181.78) mm, rotated rx -9.61 ry -16.54 rz -54.03 deg; joints [-12.301, -63.234, 112.226, 196.848, 33.775, -116.61, -415]
  MoveL 5604 to (-71.44, -25.13, -181.78) mm, rotated rx -9.61 ry -16.54 rz -54.03 deg; joints [-12.301, -63.253, 112.21, 196.864, 33.742, -116.629, -415]
  MoveL 5605 to (-71.79, -25.49, -181.77) mm, rotated rx -9.61 ry -16.54 rz -54.03 deg; joints [-12.3, -63.272, 112.196, 196.88, 33.71, -116.648, -415]
  MoveL 5606 to (-72.13, -25.86, -181.74) mm, rotated rx -9.61 ry -16.54 rz -54.03 deg; joints [-12.298, -63.291, 112.182, 196.897, 33.679, -116.667, -415]
  MoveL 5607 to (-72.49, -26.23, -181.73) mm, rotated rx -9.61 ry -16.54 rz -54.03 deg; joints [-12.297, -63.309, 112.167, 196.914, 33.647, -116.686, -415]
  MoveL 5608 to (-74.34, -28.1, -181.73) mm, rotated rx -9.61 ry -16.54 rz -54.03 deg; joints [-12.294, -63.403, 112.086, 196.996, 33.48, -116.781, -415]
  MoveL 5609 to (-75.4, -29.08, -181.81) mm, rotated rx -9.61 ry -16.54 rz -54.03 deg; joints [-12.295, -63.45, 112.035, 197.037, 33.386, -116.832, -415]
  MoveL 5610 to (-76.38, -29.79, -182.06) mm, rotated rx -9.61 ry -16.54 rz -54.03 deg; joints [-12.303, -63.479, 111.979, 197.061, 33.304, -116.868, -415]
  MoveL 5611 to (-77.25, -30.2, -182.48) mm, rotated rx -9.61 ry -16.54 rz -54.03 deg; joints [-12.317, -63.489, 111.919, 197.068, 33.234, -116.889, -415]
  MoveL 5612 to (-78.02, -30.34, -183.06) mm, rotated rx -9.61 ry -16.54 rz -54.03 deg; joints [-12.338, -63.481, 111.856, 197.058, 33.177, -116.895, -415]
  MoveL 5613 to (-78.7, -30.19, -183.81) mm, rotated rx -9.61 ry -16.54 rz -54.03 deg; joints [-12.365, -63.455, 111.788, 197.03, 33.132, -116.886, -415]
  MoveL 5614 to (-79.28, -29.76, -184.72) mm, rotated rx -9.61 ry -16.54 rz -54.03 deg; joints [-12.398, -63.41, 111.715, 196.984, 33.099, -116.861, -415]
  MoveL 5615 to (-80.15, -28.05, -187.06) mm, rotated rx -9.61 ry -16.54 rz -54.03 deg; joints [-12.484, -63.265, 111.559, 196.842, 33.071, -116.767, -415]
  MoveL 5616 to (-80.44, -25.79, -189.4) mm, rotated rx -9.61 ry -16.54 rz -54.03 deg; joints [-12.572, -63.094, 111.428, 196.673, 33.093, -116.644, -415]
  MoveL 5617 to (-79.97, -23.57, -191.11) mm, rotated rx -9.61 ry -16.54 rz -54.03 deg; joints [-12.637, -62.943, 111.366, 196.522, 33.166, -116.522, -415]
  MoveL 5618 to (-79.46, -22.48, -191.72) mm, rotated rx -9.61 ry -16.54 rz -54.03 deg; joints [-12.661, -62.874, 111.36, 196.453, 33.222, -116.461, -415]
  MoveL 5619 to (-78.75, -21.39, -192.18) mm, rotated rx -9.61 ry -16.54 rz -54.03 deg; joints [-12.68, -62.811, 111.372, 196.389, 33.29, -116.401, -415]
  MoveL 5620 to (-76.78, -19.25, -192.61) mm, rotated rx -9.61 ry -16.54 rz -54.03 deg; joints [-12.7, -62.698, 111.447, 196.273, 33.467, -116.281, -415]
  MoveL 5621 to (-76.03, -18.57, -192.64) mm, rotated rx -9.61 ry -16.54 rz -54.03 deg; joints [-12.703, -62.666, 111.482, 196.24, 33.531, -116.243, -415]
  MoveL 5622 to (-73.96, -16.96, -192.64) mm, rotated rx -9.61 ry -16.54 rz -54.03 deg; joints [-12.708, -62.592, 111.588, 196.156, 33.703, -116.147, -415]
  MoveL 5623 to (-73.2, -16.31, -192.7) mm, rotated rx -9.61 ry -16.54 rz -54.03 deg; joints [-12.712, -62.561, 111.625, 196.121, 33.767, -116.109, -415]
  MoveL 5624 to (-72.37, -15.66, -192.7) mm, rotated rx -9.61 ry -16.54 rz -54.03 deg; joints [-12.714, -62.531, 111.667, 196.087, 33.836, -116.07, -415]
  MoveL 5625 to (-71.99, -15.36, -192.71) mm, rotated rx -9.61 ry -16.54 rz -54.03 deg; joints [-12.716, -62.517, 111.686, 196.071, 33.867, -116.053, -415]
  MoveL 5626 to (-71.66, -15.08, -192.73) mm, rotated rx -9.61 ry -16.54 rz -54.03 deg; joints [-12.717, -62.504, 111.702, 196.057, 33.895, -116.036, -415]
  MoveL 5627 to (-71.3, -14.79, -192.74) mm, rotated rx -9.61 ry -16.54 rz -54.03 deg; joints [-12.719, -62.49, 111.719, 196.041, 33.925, -116.019, -415]
  MoveL 5628 to (-69.24, -13.18, -192.75) mm, rotated rx -9.61 ry -16.54 rz -54.03 deg; joints [-12.724, -62.415, 111.824, 195.959, 34.096, -115.925, -415]
  MoveL 5629 to (-68.86, -12.86, -192.77) mm, rotated rx -9.61 ry -16.54 rz -54.03 deg; joints [-12.725, -62.4, 111.842, 195.943, 34.128, -115.907, -415]
  MoveL 5630 to (-68.52, -12.54, -192.81) mm, rotated rx -9.61 ry -16.54 rz -54.03 deg; joints [-12.728, -62.384, 111.857, 195.927, 34.157, -115.889, -415]
  MoveL 5631 to (-68.22, -12.22, -192.85) mm, rotated rx -9.61 ry -16.54 rz -54.03 deg; joints [-12.73, -62.367, 111.868, 195.912, 34.184, -115.873, -415]
  MoveL 5632 to (-67.95, -11.88, -192.88) mm, rotated rx -9.61 ry -16.54 rz -54.03 deg; joints [-12.731, -62.348, 111.877, 195.898, 34.21, -115.858, -415]
  MoveL 5633 to (-67.73, -11.5, -192.9) mm, rotated rx -9.61 ry -16.54 rz -54.03 deg; joints [-12.732, -62.326, 111.88, 195.887, 34.234, -115.845, -415]
  MoveL 5634 to (-67.55, -11.09, -192.9) mm, rotated rx -9.61 ry -16.54 rz -54.03 deg; joints [-12.732, -62.302, 111.879, 195.878, 34.257, -115.834, -415]
  MoveL 5635 to (-67.98, -11.72, -193.64) mm, rotated rx -9.61 ry -16.54 rz -54.03 deg; joints [-12.762, -62.332, 111.859, 195.847, 34.204, -115.825, -415]
  MoveL 5636 to (-67.78, -10.3, -194.19) mm, rotated rx -9.61 ry -16.54 rz -54.03 deg; joints [-12.781, -62.236, 111.817, 195.794, 34.251, -115.778, -415]
  MoveL 5637 to (-67.46, -8.78, -194.62) mm, rotated rx -9.61 ry -16.54 rz -54.03 deg; joints [-12.795, -62.136, 111.78, 195.746, 34.31, -115.732, -415]
  MoveL 5638 to (-67.02, -7.06, -194.92) mm, rotated rx -9.61 ry -16.54 rz -54.03 deg; joints [-12.804, -62.027, 111.748, 195.699, 34.383, -115.684, -415]
  MoveL 5639 to (-66.43, -5.13, -195.11) mm, rotated rx -9.61 ry -16.54 rz -54.03 deg; joints [-12.808, -61.905, 111.721, 195.655, 34.473, -115.635, -415]
  MoveL 5640 to (-65.82, -3.12, -195.3) mm, rotated rx -9.61 ry -16.54 rz -54.03 deg; joints [-12.813, -61.779, 111.693, 195.609, 34.566, -115.583, -415]
  MoveL 5641 to (-65.17, -1.09, -195.42) mm, rotated rx -9.61 ry -16.54 rz -54.03 deg; joints [-12.814, -61.653, 111.667, 195.568, 34.663, -115.534, -415]
  MoveL 5642 to (-64.53, 0.94, -195.65) mm, rotated rx -9.61 ry -16.54 rz -54.03 deg; joints [-12.82, -61.525, 111.638, 195.52, 34.758, -115.481, -415]
  MoveL 5643 to (-63.87, 2.97, -195.76) mm, rotated rx -9.61 ry -16.54 rz -54.03 deg; joints [-12.822, -61.398, 111.612, 195.479, 34.854, -115.432, -415]
  MoveL 5644 to (-63.21, 5, -195.88) mm, rotated rx -9.61 ry -16.54 rz -54.03 deg; joints [-12.823, -61.271, 111.586, 195.438, 34.951, -115.384, -415]
  MoveL 5645 to (-62.55, 7.03, -196) mm, rotated rx -9.61 ry -16.54 rz -54.03 deg; joints [-12.825, -61.144, 111.559, 195.397, 35.047, -115.336, -415]
  MoveL 5646 to (-61.89, 9.06, -196.23) mm, rotated rx -9.61 ry -16.54 rz -54.03 deg; joints [-12.831, -61.017, 111.531, 195.35, 35.142, -115.283, -415]
  MoveL 5647 to (-61.23, 11.09, -196.35) mm, rotated rx -9.61 ry -16.54 rz -54.03 deg; joints [-12.832, -60.89, 111.504, 195.309, 35.238, -115.236, -415]
  MoveL 5648 to (-60.64, 13.06, -196.46) mm, rotated rx -9.61 ry -16.54 rz -54.03 deg; joints [-12.833, -60.766, 111.472, 195.274, 35.327, -115.193, -415]
  MoveL 5649 to (-60.18, 15.02, -196.66) mm, rotated rx -9.61 ry -16.54 rz -54.03 deg; joints [-12.838, -60.64, 111.431, 195.235, 35.408, -115.15, -415]
  MoveL 5650 to (-59.37, 17.38, -196.8) mm, rotated rx -9.61 ry -16.54 rz -54.03 deg; joints [-12.84, -60.491, 111.4, 195.189, 35.521, -115.094, -415]
  MoveL 5651 to (-58.46, 19.66, -196.88) mm, rotated rx -9.61 ry -16.54 rz -54.03 deg; joints [-12.84, -60.351, 111.382, 195.143, 35.639, -115.039, -415]
  MoveL 5652 to (-57.67, 21.81, -196.92) mm, rotated rx -9.61 ry -16.54 rz -54.03 deg; joints [-12.838, -60.218, 111.359, 195.106, 35.746, -114.991, -415]
  MoveL 5653 to (-57.01, 23.75, -196.96) mm, rotated rx -9.61 ry -16.54 rz -54.03 deg; joints [-12.837, -60.096, 111.333, 195.073, 35.839, -114.95, -415]
  MoveL 5654 to (-56.39, 25.61, -197.08) mm, rotated rx -9.61 ry -16.54 rz -54.03 deg; joints [-12.839, -59.979, 111.307, 195.037, 35.926, -114.908, -415]
  MoveL 5655 to (-55.76, 27.53, -197.14) mm, rotated rx -9.61 ry -16.54 rz -54.03 deg; joints [-12.839, -59.858, 111.28, 195.005, 36.016, -114.867, -415]
  MoveL 5656 to (-55.08, 29.55, -197.22) mm, rotated rx -9.61 ry -16.54 rz -54.03 deg; joints [-12.839, -59.732, 111.251, 194.97, 36.111, -114.824, -415]
  MoveL 5657 to (-54.43, 31.43, -197.4) mm, rotated rx -9.61 ry -16.54 rz -54.03 deg; joints [-12.843, -59.613, 111.225, 194.93, 36.2, -114.779, -415]
  MoveL 5658 to (-53.78, 33.22, -197.71) mm, rotated rx -9.61 ry -16.54 rz -54.03 deg; joints [-12.853, -59.499, 111.2, 194.883, 36.284, -114.73, -415]
  MoveL 5659 to (-53.11, 33.78, -198.75) mm, rotated rx -9.61 ry -16.54 rz -54.03 deg; joints [-12.897, -59.463, 111.215, 194.795, 36.327, -114.664, -415]
  MoveL 5660 to (-53.14, 33.52, -199.27) mm, rotated rx -9.61 ry -16.54 rz -54.03 deg; joints [-12.918, -59.476, 111.217, 194.765, 36.312, -114.647, -415]
  MoveL 5661 to (-53.12, 33.5, -199.59) mm, rotated rx -9.61 ry -16.54 rz -54.03 deg; joints [-12.932, -59.476, 111.215, 194.744, 36.309, -114.634, -415]
  MoveL 5662 to (-53.07, 33.71, -199.76) mm, rotated rx -9.61 ry -16.54 rz -54.03 deg; joints [-12.938, -59.461, 111.208, 194.731, 36.316, -114.624, -415]
  MoveL 5663 to (-53.04, 34.14, -199.79) mm, rotated rx -9.61 ry -16.54 rz -54.03 deg; joints [-12.938, -59.433, 111.193, 194.726, 36.328, -114.618, -415]
  MoveL 5664 to (-53.05, 34.65, -199.81) mm, rotated rx -9.61 ry -16.54 rz -54.03 deg; joints [-12.937, -59.398, 111.171, 194.724, 36.341, -114.614, -415]
  MoveL 5665 to (-53.15, 35.24, -199.82) mm, rotated rx -9.61 ry -16.54 rz -54.03 deg; joints [-12.935, -59.357, 111.14, 194.723, 36.35, -114.612, -415]
  MoveL 5666 to (-53.29, 35.86, -199.83) mm, rotated rx -9.61 ry -16.54 rz -54.03 deg; joints [-12.933, -59.314, 111.104, 194.724, 36.358, -114.611, -415]
  MoveL 5667 to (-54.27, 39.39, -199.83) mm, rotated rx -9.61 ry -16.54 rz -54.03 deg; joints [-12.916, -59.064, 110.885, 194.74, 36.39, -114.614, -415]
  MoveL 5668 to (-54.38, 39.82, -199.86) mm, rotated rx -9.61 ry -16.54 rz -54.03 deg; joints [-12.916, -59.034, 110.86, 194.74, 36.395, -114.613, -415]
  MoveL 5669 to (-54.5, 40.29, -199.87) mm, rotated rx -9.61 ry -16.54 rz -54.03 deg; joints [-12.914, -59.001, 110.831, 194.741, 36.399, -114.613, -415]
  MoveL 5670 to (-54.64, 40.79, -199.88) mm, rotated rx -9.61 ry -16.54 rz -54.03 deg; joints [-12.912, -58.965, 110.8, 194.743, 36.404, -114.613, -415]
  MoveL 5671 to (-54.76, 41.27, -199.89) mm, rotated rx -9.61 ry -16.54 rz -54.03 deg; joints [-12.91, -58.932, 110.771, 194.743, 36.409, -114.613, -415]
  MoveL 5672 to (-54.86, 41.72, -199.93) mm, rotated rx -9.61 ry -16.54 rz -54.03 deg; joints [-12.91, -58.9, 110.744, 194.742, 36.414, -114.611, -415]
  MoveL 5673 to (-54.93, 42.14, -199.99) mm, rotated rx -9.61 ry -16.54 rz -54.03 deg; joints [-12.911, -58.87, 110.72, 194.739, 36.42, -114.608, -415]
  MoveL 5674 to (-55.04, 42.6, -200.03) mm, rotated rx -9.61 ry -16.54 rz -54.03 deg; joints [-12.91, -58.838, 110.693, 194.738, 36.425, -114.606, -415]
  MoveL 5675 to (-55.15, 43.08, -200.04) mm, rotated rx -9.61 ry -16.54 rz -54.03 deg; joints [-12.909, -58.804, 110.665, 194.739, 36.429, -114.605, -415]
  MoveL 5676 to (-55.29, 43.56, -200.05) mm, rotated rx -9.61 ry -16.54 rz -54.03 deg; joints [-12.907, -58.77, 110.634, 194.741, 36.434, -114.606, -415]
  MoveL 5677 to (-55.43, 44.07, -200.05) mm, rotated rx -9.61 ry -16.54 rz -54.03 deg; joints [-12.904, -58.734, 110.603, 194.743, 36.438, -114.606, -415]
  MoveL 5678 to (-55.93, 46.94, -200.39) mm, rotated rx -9.61 ry -16.54 rz -54.03 deg; joints [-12.906, -58.533, 110.442, 194.726, 36.477, -114.587, -415]
  MoveL 5679 to (-55.92, 48.24, -200.83) mm, rotated rx -9.61 ry -16.54 rz -54.03 deg; joints [-12.92, -58.443, 110.384, 194.694, 36.505, -114.56, -415]
  MoveL 5680 to (-55.73, 49.45, -201.43) mm, rotated rx -9.61 ry -16.54 rz -54.03 deg; joints [-12.941, -58.36, 110.34, 194.646, 36.541, -114.522, -415]
  MoveL 5681 to (-54.82, 51.6, -203.16) mm, rotated rx -9.61 ry -16.54 rz -54.03 deg; joints [-13.008, -58.216, 110.299, 194.505, 36.63, -114.411, -415]
  MoveL 5682 to (-53.22, 53.38, -205.59) mm, rotated rx -9.61 ry -16.54 rz -54.03 deg; joints [-13.107, -58.099, 110.318, 194.302, 36.745, -114.257, -415]
  MoveL 5683 to (-51.44, 54.38, -208.01) mm, rotated rx -9.61 ry -16.54 rz -54.03 deg; joints [-13.21, -58.037, 110.38, 194.099, 36.852, -114.104, -415]
  MoveL 5684 to (-50.7, 54.44, -208.96) mm, rotated rx -9.61 ry -16.54 rz -54.03 deg; joints [-13.251, -58.035, 110.423, 194.018, 36.888, -114.045, -415]
  MoveL 5685 to (-50.05, 54.2, -209.74) mm, rotated rx -9.61 ry -16.54 rz -54.03 deg; joints [-13.287, -58.053, 110.472, 193.952, 36.914, -113.997, -415]
  MoveL 5686 to (-49.76, 53.97, -210.06) mm, rotated rx -9.61 ry -16.54 rz -54.03 deg; joints [-13.302, -58.07, 110.5, 193.925, 36.922, -113.978, -415]
  MoveL 5687 to (-49.49, 53.67, -210.35) mm, rotated rx -9.61 ry -16.54 rz -54.03 deg; joints [-13.316, -58.091, 110.529, 193.901, 36.928, -113.961, -415]
  MoveL 5688 to (-49.02, 52.84, -210.78) mm, rotated rx -9.61 ry -16.54 rz -54.03 deg; joints [-13.338, -58.15, 110.594, 193.863, 36.931, -113.936, -415]
  MoveL 5689 to (-48.65, 51.71, -211.04) mm, rotated rx -9.61 ry -16.54 rz -54.03 deg; joints [-13.354, -58.228, 110.666, 193.839, 36.922, -113.923, -415]
  MoveL 5690 to (-48.37, 50.29, -211.12) mm, rotated rx -9.61 ry -16.54 rz -54.03 deg; joints [-13.364, -58.326, 110.745, 193.83, 36.902, -113.921, -415]
  MoveL 5691 to (-48.3, 49.77, -211.12) mm, rotated rx -9.61 ry -16.54 rz -54.03 deg; joints [-13.366, -58.362, 110.773, 193.829, 36.894, -113.922, -415]
  MoveL 5692 to (-48.25, 49.32, -211.1) mm, rotated rx -9.61 ry -16.54 rz -54.03 deg; joints [-13.367, -58.393, 110.795, 193.831, 36.885, -113.925, -415]
  MoveL 5693 to (-48.22, 48.89, -211.05) mm, rotated rx -9.61 ry -16.54 rz -54.03 deg; joints [-13.367, -58.422, 110.816, 193.834, 36.877, -113.928, -415]
  MoveL 5694 to (-48.2, 48.47, -210.99) mm, rotated rx -9.61 ry -16.54 rz -54.03 deg; joints [-13.366, -58.451, 110.835, 193.838, 36.868, -113.933, -415]
  MoveL 5695 to (-48.17, 48.02, -210.95) mm, rotated rx -9.61 ry -16.54 rz -54.03 deg; joints [-13.366, -58.482, 110.857, 193.841, 36.859, -113.936, -415]
  MoveL 5696 to (-48.11, 47.51, -210.94) mm, rotated rx -9.61 ry -16.54 rz -54.03 deg; joints [-13.367, -58.517, 110.883, 193.842, 36.85, -113.939, -415]
  MoveL 5697 to (-48.03, 47, -210.94) mm, rotated rx -9.61 ry -16.54 rz -54.03 deg; joints [-13.37, -58.553, 110.91, 193.841, 36.841, -113.94, -415]
  MoveL 5698 to (-47.96, 46.5, -210.93) mm, rotated rx -9.61 ry -16.54 rz -54.03 deg; joints [-13.371, -58.587, 110.936, 193.841, 36.833, -113.941, -415]
  MoveL 5699 to (-47.9, 46.03, -210.91) mm, rotated rx -9.61 ry -16.54 rz -54.03 deg; joints [-13.372, -58.619, 110.96, 193.842, 36.825, -113.944, -415]
  MoveL 5700 to (-47.87, 45.61, -210.85) mm, rotated rx -9.61 ry -16.54 rz -54.03 deg; joints [-13.372, -58.649, 110.981, 193.845, 36.817, -113.948, -415]
  MoveL 5701 to (-47.84, 45.19, -210.79) mm, rotated rx -9.61 ry -16.54 rz -54.03 deg; joints [-13.371, -58.678, 111.001, 193.849, 36.808, -113.952, -415]
  MoveL 5702 to (-47.81, 44.72, -210.74) mm, rotated rx -9.61 ry -16.54 rz -54.03 deg; joints [-13.371, -58.71, 111.024, 193.853, 36.799, -113.956, -415]
  MoveL 5703 to (-47.74, 44.11, -210.7) mm, rotated rx -9.61 ry -16.54 rz -54.03 deg; joints [-13.372, -58.752, 111.054, 193.855, 36.787, -113.96, -415]
  MoveL 5704 to (-47.66, 43.33, -210.68) mm, rotated rx -9.61 ry -16.54 rz -54.03 deg; joints [-13.374, -58.806, 111.093, 193.857, 36.773, -113.964, -415]
  MoveL 5705 to (-47.43, 41.77, -210.68) mm, rotated rx -9.61 ry -16.54 rz -54.03 deg; joints [-13.38, -58.913, 111.174, 193.855, 36.746, -113.968, -415]
  MoveL 5706 to (-47.32, 40.94, -210.65) mm, rotated rx -9.61 ry -16.54 rz -54.03 deg; joints [-13.383, -58.97, 111.217, 193.856, 36.732, -113.971, -415]
  MoveL 5707 to (-47.24, 40.32, -210.64) mm, rotated rx -9.61 ry -16.54 rz -54.03 deg; joints [-13.385, -59.013, 111.248, 193.856, 36.72, -113.974, -415]
  MoveL 5708 to (-47.22, 39.83, -210.63) mm, rotated rx -9.61 ry -16.54 rz -54.03 deg; joints [-13.386, -59.046, 111.27, 193.858, 36.709, -113.977, -415]
  MoveL 5709 to (-47.24, 39.42, -210.61) mm, rotated rx -9.61 ry -16.54 rz -54.03 deg; joints [-13.387, -59.074, 111.286, 193.861, 36.697, -113.981, -415]
  MoveL 5710 to (-47.29, 39.22, -210.5) mm, rotated rx -9.61 ry -16.54 rz -54.03 deg; joints [-13.383, -59.088, 111.291, 193.87, 36.69, -113.989, -415]
  MoveL 5711 to (-47.33, 39.28, -210.28) mm, rotated rx -9.61 ry -16.54 rz -54.03 deg; joints [-13.373, -59.085, 111.288, 193.884, 36.692, -113.998, -415]
  MoveL 5712 to (-47.35, 39.61, -209.93) mm, rotated rx -9.61 ry -16.54 rz -54.03 deg; joints [-13.358, -59.064, 111.278, 193.905, 36.704, -114.009, -415]
  MoveL 5713 to (-48.05, 39.27, -209.23) mm, rotated rx -9.61 ry -16.54 rz -54.03 deg; joints [-13.327, -59.084, 111.248, 193.971, 36.66, -114.06, -415]
  MoveL 5714 to (-48.95, 37.47, -209.08) mm, rotated rx -9.61 ry -16.54 rz -54.03 deg; joints [-13.323, -59.194, 111.253, 194.012, 36.558, -114.107, -415]
  MoveL 5715 to (-49.84, 35.77, -208.8) mm, rotated rx -9.61 ry -16.54 rz -54.03 deg; joints [-13.312, -59.3, 111.257, 194.062, 36.461, -114.159, -415]
  MoveL 5716 to (-50.72, 34.05, -208.52) mm, rotated rx -9.61 ry -16.54 rz -54.03 deg; joints [-13.303, -59.406, 111.262, 194.111, 36.365, -114.21, -415]
  MoveL 5717 to (-51.59, 32.32, -208.25) mm, rotated rx -9.61 ry -16.54 rz -54.03 deg; joints [-13.293, -59.513, 111.267, 194.16, 36.268, -114.261, -415]
  MoveL 5718 to (-52.5, 30.51, -208.04) mm, rotated rx -9.61 ry -16.54 rz -54.03 deg; joints [-13.286, -59.624, 111.272, 194.207, 36.166, -114.313, -415]
  MoveL 5719 to (-53.5, 28.64, -207.89) mm, rotated rx -9.61 ry -16.54 rz -54.03 deg; joints [-13.281, -59.737, 111.271, 194.253, 36.056, -114.366, -415]
  MoveL 5720 to (-54.8, 26.46, -207.79) mm, rotated rx -9.61 ry -16.54 rz -54.03 deg; joints [-13.277, -59.867, 111.258, 194.307, 35.918, -114.429, -415]
  MoveL 5721 to (-55.75, 24.16, -207.71) mm, rotated rx -9.61 ry -16.54 rz -54.03 deg; joints [-13.277, -60.009, 111.276, 194.35, 35.798, -114.482, -415]
  MoveL 5722 to (-56.56, 22.21, -207.6) mm, rotated rx -9.61 ry -16.54 rz -54.03 deg; joints [-13.275, -60.129, 111.291, 194.39, 35.696, -114.529, -415]
  MoveL 5723 to (-57.33, 20.48, -207.42) mm, rotated rx -9.61 ry -16.54 rz -54.03 deg; joints [-13.27, -60.236, 111.301, 194.432, 35.603, -114.576, -415]
  MoveL 5724 to (-58.2, 18.64, -207.29) mm, rotated rx -9.61 ry -16.54 rz -54.03 deg; joints [-13.266, -60.348, 111.307, 194.475, 35.501, -114.625, -415]
  MoveL 5725 to (-59.09, 16.75, -207.16) mm, rotated rx -9.61 ry -16.54 rz -54.03 deg; joints [-13.263, -60.463, 111.312, 194.519, 35.396, -114.676, -415]
  MoveL 5726 to (-60.02, 14.79, -207.09) mm, rotated rx -9.61 ry -16.54 rz -54.03 deg; joints [-13.262, -60.581, 111.316, 194.561, 35.285, -114.726, -415]
  MoveL 5727 to (-60.93, 12.86, -206.87) mm, rotated rx -9.61 ry -16.54 rz -54.03 deg; joints [-13.255, -60.699, 111.323, 194.613, 35.178, -114.783, -415]
  MoveL 5728 to (-61.84, 10.93, -206.75) mm, rotated rx -9.61 ry -16.54 rz -54.03 deg; joints [-13.252, -60.816, 111.327, 194.658, 35.07, -114.835, -415]
  MoveL 5729 to (-62.73, 8.99, -206.53) mm, rotated rx -9.61 ry -16.54 rz -54.03 deg; joints [-13.245, -60.934, 111.334, 194.71, 34.963, -114.892, -415]
  MoveL 5730 to (-63.64, 7.05, -206.42) mm, rotated rx -9.61 ry -16.54 rz -54.03 deg; joints [-13.242, -61.051, 111.338, 194.755, 34.855, -114.945, -415]
  MoveL 5731 to (-64.52, 5.11, -206.2) mm, rotated rx -9.61 ry -16.54 rz -54.03 deg; joints [-13.235, -61.17, 111.345, 194.807, 34.748, -115.002, -415]
  MoveL 5732 to (-65.42, 3.18, -206.09) mm, rotated rx -9.61 ry -16.54 rz -54.03 deg; joints [-13.233, -61.286, 111.349, 194.853, 34.64, -115.055, -415]
  MoveL 5733 to (-66.32, 1.24, -205.99) mm, rotated rx -9.61 ry -16.54 rz -54.03 deg; joints [-13.23, -61.403, 111.353, 194.899, 34.531, -115.109, -415]
  MoveL 5734 to (-67.07, -0.53, -205.75) mm, rotated rx -9.61 ry -16.54 rz -54.03 deg; joints [-13.223, -61.511, 111.363, 194.948, 34.438, -115.162, -415]
  MoveL 5735 to (-67.75, -2.22, -205.45) mm, rotated rx -9.61 ry -16.54 rz -54.03 deg; joints [-13.213, -61.616, 111.377, 194.999, 34.351, -115.214, -415]
  MoveL 5736 to (-68.37, -3.91, -205.06) mm, rotated rx -9.61 ry -16.54 rz -54.03 deg; joints [-13.2, -61.721, 111.395, 195.055, 34.269, -115.269, -415]
  MoveL 5737 to (-67.52, -2.77, -204.14) mm, rotated rx -9.61 ry -16.54 rz -54.03 deg; joints [-13.163, -61.666, 111.432, 195.082, 34.365, -115.268, -415]
  MoveL 5738 to (-67.69, -3.1, -204.08) mm, rotated rx -9.61 ry -16.54 rz -54.03 deg; joints [-13.16, -61.685, 111.432, 195.093, 34.346, -115.279, -415]
  MoveL 5739 to (-67.88, -3.42, -204.03) mm, rotated rx -9.61 ry -16.54 rz -54.03 deg; joints [-13.158, -61.704, 111.429, 195.105, 34.326, -115.291, -415]
  MoveL 5740 to (-68.16, -3.72, -203.99) mm, rotated rx -9.61 ry -16.54 rz -54.03 deg; joints [-13.156, -61.72, 111.419, 195.118, 34.301, -115.306, -415]
  MoveL 5741 to (-68.5, -4.02, -203.97) mm, rotated rx -9.61 ry -16.54 rz -54.03 deg; joints [-13.155, -61.735, 111.403, 195.132, 34.272, -115.322, -415]
  MoveL 5742 to (-68.92, -4.3, -203.96) mm, rotated rx -9.61 ry -16.54 rz -54.03 deg; joints [-13.153, -61.747, 111.381, 195.148, 34.238, -115.339, -415]
  MoveL 5743 to (-69.36, -4.57, -203.96) mm, rotated rx -9.61 ry -16.54 rz -54.03 deg; joints [-13.152, -61.758, 111.357, 195.164, 34.204, -115.358, -415]
  MoveL 5744 to (-70.26, -5.11, -203.95) mm, rotated rx -9.61 ry -16.54 rz -54.03 deg; joints [-13.149, -61.78, 111.305, 195.198, 34.134, -115.395, -415]
  MoveL 5745 to (-70.67, -5.37, -203.94) mm, rotated rx -9.61 ry -16.54 rz -54.03 deg; joints [-13.147, -61.791, 111.283, 195.214, 34.102, -115.413, -415]
  MoveL 5746 to (-71.06, -5.64, -203.89) mm, rotated rx -9.61 ry -16.54 rz -54.03 deg; joints [-13.144, -61.804, 111.263, 195.232, 34.072, -115.431, -415]
  MoveL 5747 to (-71.48, -5.95, -203.81) mm, rotated rx -9.61 ry -16.54 rz -54.03 deg; joints [-13.139, -61.818, 111.242, 195.253, 34.038, -115.453, -415]
  MoveL 5748 to (-71.96, -6.28, -203.75) mm, rotated rx -9.61 ry -16.54 rz -54.03 deg; joints [-13.136, -61.833, 111.217, 195.275, 34, -115.476, -415]
  MoveL 5749 to (-72.44, -6.59, -203.71) mm, rotated rx -9.61 ry -16.54 rz -54.03 deg; joints [-13.133, -61.847, 111.191, 195.295, 33.963, -115.498, -415]
  MoveL 5750 to (-72.9, -6.88, -203.7) mm, rotated rx -9.61 ry -16.54 rz -54.03 deg; joints [-13.131, -61.858, 111.165, 195.313, 33.927, -115.518, -415]
  MoveL 5751 to (-73.36, -7.15, -203.7) mm, rotated rx -9.61 ry -16.54 rz -54.03 deg; joints [-13.129, -61.869, 111.139, 195.33, 33.891, -115.537, -415]
  MoveL 5752 to (-74.26, -7.69, -203.7) mm, rotated rx -9.61 ry -16.54 rz -54.03 deg; joints [-13.126, -61.89, 111.087, 195.364, 33.821, -115.575, -415]
  MoveL 5753 to (-75.13, -8.24, -203.67) mm, rotated rx -9.61 ry -16.54 rz -54.03 deg; joints [-13.123, -61.914, 111.039, 195.398, 33.753, -115.613, -415]
  MoveL 5754 to (-77.38, -9.58, -203.67) mm, rotated rx -9.61 ry -16.54 rz -54.03 deg; joints [-13.116, -61.966, 110.91, 195.483, 33.579, -115.709, -415]
  MoveL 5755 to (-78.65, -10.26, -203.76) mm, rotated rx -9.61 ry -16.54 rz -54.03 deg; joints [-13.115, -61.99, 110.832, 195.525, 33.482, -115.758, -415]
  MoveL 5756 to (-79.76, -10.68, -204.02) mm, rotated rx -9.61 ry -16.54 rz -54.03 deg; joints [-13.121, -61.997, 110.756, 195.548, 33.4, -115.792, -415]
  MoveL 5757 to (-80.68, -10.84, -204.46) mm, rotated rx -9.61 ry -16.54 rz -54.03 deg; joints [-13.135, -61.989, 110.682, 195.552, 33.334, -115.808, -415]
  MoveL 5758 to (-81.08, -10.82, -204.75) mm, rotated rx -9.61 ry -16.54 rz -54.03 deg; joints [-13.144, -61.979, 110.646, 195.546, 33.307, -115.81, -415]
  MoveL 5759 to (-81.44, -10.74, -205.08) mm, rotated rx -9.61 ry -16.54 rz -54.03 deg; joints [-13.155, -61.966, 110.611, 195.536, 33.284, -115.808, -415]
  MoveL 5760 to (-82.01, -10.37, -205.86) mm, rotated rx -9.61 ry -16.54 rz -54.03 deg; joints [-13.183, -61.926, 110.541, 195.5, 33.251, -115.79, -415]
  MoveL 5761 to (-82.42, -9.75, -206.83) mm, rotated rx -9.61 ry -16.54 rz -54.03 deg; joints [-13.218, -61.871, 110.474, 195.445, 33.233, -115.756, -415]
  MoveL 5762 to (-82.7, -7.72, -209.29) mm, rotated rx -9.61 ry -16.54 rz -54.03 deg; joints [-13.309, -61.714, 110.345, 195.277, 33.244, -115.636, -415]
  MoveL 5763 to (-82.27, -5.33, -211.74) mm, rotated rx -9.61 ry -16.54 rz -54.03 deg; joints [-13.402, -61.544, 110.258, 195.084, 33.308, -115.489, -415]
  MoveL 5764 to (-81.14, -3.26, -213.5) mm, rotated rx -9.61 ry -16.54 rz -54.03 deg; joints [-13.471, -61.412, 110.248, 194.917, 33.414, -115.351, -415]
  MoveL 5765 to (-80.3, -2.35, -214.11) mm, rotated rx -9.61 ry -16.54 rz -54.03 deg; joints [-13.497, -61.36, 110.272, 194.843, 33.483, -115.285, -415]
  MoveL 5766 to (-79.29, -1.51, -214.55) mm, rotated rx -9.61 ry -16.54 rz -54.03 deg; joints [-13.517, -61.318, 110.315, 194.775, 33.562, -115.223, -415]
  MoveL 5767 to (-76.74, -0.08, -214.9) mm, rotated rx -9.61 ry -16.54 rz -54.03 deg; joints [-13.54, -61.261, 110.46, 194.659, 33.753, -115.104, -415]
  MoveL 5768 to (-74.33, 0.97, -214.9) mm, rotated rx -9.61 ry -16.54 rz -54.03 deg; joints [-13.549, -61.229, 110.611, 194.575, 33.929, -115.011, -415]
  MoveL 5769 to (-73.84, 1.17, -214.89) mm, rotated rx -9.61 ry -16.54 rz -54.03 deg; joints [-13.551, -61.223, 110.642, 194.559, 33.965, -114.993, -415]
  MoveL 5770 to (-73.34, 1.37, -214.85) mm, rotated rx -9.61 ry -16.54 rz -54.03 deg; joints [-13.552, -61.218, 110.675, 194.543, 34.001, -114.975, -415]
  MoveL 5771 to (-72.88, 1.57, -214.85) mm, rotated rx -9.61 ry -16.54 rz -54.03 deg; joints [-13.553, -61.212, 110.704, 194.528, 34.035, -114.958, -415]
  MoveL 5772 to (-72.48, 1.75, -214.86) mm, rotated rx -9.61 ry -16.54 rz -54.03 deg; joints [-13.555, -61.206, 110.729, 194.513, 34.064, -114.941, -415]
  MoveL 5773 to (-72.03, 1.96, -214.89) mm, rotated rx -9.61 ry -16.54 rz -54.03 deg; joints [-13.558, -61.199, 110.755, 194.496, 34.097, -114.923, -415]
  MoveL 5774 to (-71.52, 2.24, -214.96) mm, rotated rx -9.61 ry -16.54 rz -54.03 deg; joints [-13.562, -61.188, 110.785, 194.473, 34.135, -114.9, -415]
  MoveL 5775 to (-71.02, 2.51, -215.04) mm, rotated rx -9.61 ry -16.54 rz -54.03 deg; joints [-13.567, -61.177, 110.813, 194.45, 34.172, -114.877, -415]
  MoveL 5776 to (-70.51, 2.77, -215.09) mm, rotated rx -9.61 ry -16.54 rz -54.03 deg; joints [-13.571, -61.167, 110.843, 194.429, 34.21, -114.855, -415]
  MoveL 5777 to (-70.03, 3, -215.11) mm, rotated rx -9.61 ry -16.54 rz -54.03 deg; joints [-13.574, -61.159, 110.872, 194.411, 34.245, -114.836, -415]
  MoveL 5778 to (-69.56, 3.21, -215.12) mm, rotated rx -9.61 ry -16.54 rz -54.03 deg; joints [-13.576, -61.152, 110.901, 194.395, 34.28, -114.818, -415]
  MoveL 5779 to (-69.08, 3.42, -215.12) mm, rotated rx -9.61 ry -16.54 rz -54.03 deg; joints [-13.578, -61.145, 110.931, 194.378, 34.315, -114.799, -415]
  MoveL 5780 to (-68.57, 3.67, -215.15) mm, rotated rx -9.61 ry -16.54 rz -54.03 deg; joints [-13.581, -61.136, 110.961, 194.358, 34.352, -114.779, -415]
  MoveL 5781 to (-68.08, 3.93, -215.2) mm, rotated rx -9.61 ry -16.54 rz -54.03 deg; joints [-13.585, -61.126, 110.989, 194.338, 34.389, -114.758, -415]
  MoveL 5782 to (-67.6, 4.21, -215.27) mm, rotated rx -9.61 ry -16.54 rz -54.03 deg; joints [-13.589, -61.114, 111.015, 194.317, 34.425, -114.736, -415]
  MoveL 5783 to (-67.19, 4.51, -215.33) mm, rotated rx -9.61 ry -16.54 rz -54.03 deg; joints [-13.593, -61.1, 111.035, 194.299, 34.458, -114.717, -415]
  MoveL 5784 to (-66.84, 4.81, -215.36) mm, rotated rx -9.61 ry -16.54 rz -54.03 deg; joints [-13.595, -61.084, 111.05, 194.284, 34.487, -114.701, -415]
  MoveL 5785 to (-66.59, 5.13, -215.37) mm, rotated rx -9.61 ry -16.54 rz -54.03 deg; joints [-13.596, -61.067, 111.059, 194.274, 34.512, -114.69, -415]
  MoveL 5786 to (-66.37, 5.45, -215.37) mm, rotated rx -9.61 ry -16.54 rz -54.03 deg; joints [-13.596, -61.049, 111.064, 194.266, 34.534, -114.679, -415]
  MoveL 5787 to (-67.23, 4.49, -216.25) mm, rotated rx -9.61 ry -16.54 rz -54.03 deg; joints [-13.63, -61.093, 111.02, 194.24, 34.443, -114.68, -415]
  MoveL 5788 to (-66.47, 5.9, -216.53) mm, rotated rx -9.61 ry -16.54 rz -54.03 deg; joints [-13.64, -61.009, 111.022, 194.191, 34.526, -114.631, -415]
  MoveL 5789 to (-65.57, 7.46, -216.73) mm, rotated rx -9.61 ry -16.54 rz -54.03 deg; joints [-13.647, -60.917, 111.032, 194.143, 34.624, -114.579, -415]
  MoveL 5790 to (-64.5, 9.21, -216.86) mm, rotated rx -9.61 ry -16.54 rz -54.03 deg; joints [-13.652, -60.815, 111.047, 194.094, 34.737, -114.523, -415]
  MoveL 5791 to (-63.3, 11.12, -216.95) mm, rotated rx -9.61 ry -16.54 rz -54.03 deg; joints [-13.656, -60.704, 111.067, 194.043, 34.862, -114.464, -415]
  MoveL 5792 to (-62.18, 12.93, -217.1) mm, rotated rx -9.61 ry -16.54 rz -54.03 deg; joints [-13.661, -60.598, 111.083, 193.991, 34.98, -114.407, -415]
  MoveL 5793 to (-61.06, 14.76, -217.31) mm, rotated rx -9.61 ry -16.54 rz -54.03 deg; joints [-13.669, -60.491, 111.097, 193.936, 35.097, -114.347, -415]
  MoveL 5794 to (-59.99, 16.48, -217.43) mm, rotated rx -9.61 ry -16.54 rz -54.03 deg; joints [-13.674, -60.39, 111.112, 193.889, 35.209, -114.294, -415]
  MoveL 5795 to (-59.04, 18.06, -217.69) mm, rotated rx -9.61 ry -16.54 rz -54.03 deg; joints [-13.684, -60.296, 111.122, 193.837, 35.308, -114.24, -415]
  MoveL 5796 to (-57.95, 19.82, -217.91) mm, rotated rx -9.61 ry -16.54 rz -54.03 deg; joints [-13.693, -60.192, 111.136, 193.783, 35.421, -114.182, -415]
  MoveL 5797 to (-56.84, 21.58, -218.05) mm, rotated rx -9.61 ry -16.54 rz -54.03 deg; joints [-13.698, -60.088, 111.151, 193.735, 35.536, -114.128, -415]
  MoveL 5798 to (-55.69, 23.38, -218.15) mm, rotated rx -9.61 ry -16.54 rz -54.03 deg; joints [-13.702, -59.982, 111.168, 193.688, 35.654, -114.074, -415]
  MoveL 5799 to (-54.57, 25.18, -218.38) mm, rotated rx -9.61 ry -16.54 rz -54.03 deg; joints [-13.711, -59.876, 111.182, 193.634, 35.77, -114.016, -415]
  MoveL 5800 to (-53.4, 26.98, -218.64) mm, rotated rx -9.61 ry -16.54 rz -54.03 deg; joints [-13.721, -59.769, 111.197, 193.577, 35.888, -113.956, -415]
  MoveL 5801 to (-52.25, 28.77, -218.73) mm, rotated rx -9.61 ry -16.54 rz -54.03 deg; joints [-13.725, -59.663, 111.214, 193.532, 36.006, -113.903, -415]
  MoveL 5802 to (-51.08, 30.6, -218.77) mm, rotated rx -9.61 ry -16.54 rz -54.03 deg; joints [-13.726, -59.555, 111.231, 193.489, 36.127, -113.852, -415]
  MoveL 5803 to (-49.94, 32.38, -218.88) mm, rotated rx -9.61 ry -16.54 rz -54.03 deg; joints [-13.73, -59.45, 111.247, 193.444, 36.245, -113.8, -415]
  MoveL 5804 to (-48.78, 34.16, -219.08) mm, rotated rx -9.61 ry -16.54 rz -54.03 deg; joints [-13.738, -59.344, 111.263, 193.393, 36.361, -113.744, -415]
  MoveL 5805 to (-47.64, 35.89, -219.42) mm, rotated rx -9.61 ry -16.54 rz -54.03 deg; joints [-13.752, -59.24, 111.276, 193.334, 36.474, -113.685, -415]
  MoveL 5806 to (-46.43, 37.68, -219.67) mm, rotated rx -9.61 ry -16.54 rz -54.03 deg; joints [-13.762, -59.133, 111.293, 193.279, 36.593, -113.626, -415]
  MoveL 5807 to (-45.24, 39.45, -219.88) mm, rotated rx -9.61 ry -16.54 rz -54.03 deg; joints [-13.771, -59.027, 111.31, 193.228, 36.712, -113.571, -415]
  MoveL 5808 to (-44.02, 41.25, -220.11) mm, rotated rx -9.61 ry -16.54 rz -54.03 deg; joints [-13.781, -58.919, 111.327, 193.174, 36.832, -113.513, -415]
  MoveL 5809 to (-42.83, 43.04, -220.26) mm, rotated rx -9.61 ry -16.54 rz -54.03 deg; joints [-13.786, -58.812, 111.343, 193.127, 36.952, -113.461, -415]
  MoveL 5810 to (-41.68, 44.82, -220.28) mm, rotated rx -9.61 ry -16.54 rz -54.03 deg; joints [-13.787, -58.705, 111.358, 193.09, 37.069, -113.415, -415]
  MoveL 5811 to (-41.09, 45.06, -220.94) mm, rotated rx -9.61 ry -16.54 rz -54.03 deg; joints [-13.816, -58.691, 111.384, 193.032, 37.104, -113.371, -415]
  MoveL 5812 to (-41.2, 44.74, -221.27) mm, rotated rx -9.61 ry -16.54 rz -54.03 deg; joints [-13.83, -58.709, 111.384, 193.015, 37.086, -113.364, -415]
  MoveL 5813 to (-41.2, 44.7, -221.48) mm, rotated rx -9.61 ry -16.54 rz -54.03 deg; joints [-13.839, -58.71, 111.383, 193.003, 37.082, -113.357, -415]
  MoveL 5814 to (-41.13, 44.9, -221.58) mm, rotated rx -9.61 ry -16.54 rz -54.03 deg; joints [-13.842, -58.696, 111.378, 192.994, 37.09, -113.349, -415]
  MoveL 5815 to (-41.05, 45.32, -221.6) mm, rotated rx -9.61 ry -16.54 rz -54.03 deg; joints [-13.842, -58.669, 111.367, 192.99, 37.106, -113.344, -415]
  MoveC 5816 to (-41.01, 46.33, -221.6) mm, rotated rx -9.61 ry -16.54 rz -54.03 deg; joints [-13.839, -58.601, 111.329, 192.986, 37.135, -113.336, -415] to (-41.03, 47.35, -221.6) mm, rotated rx -9.61 ry -16.54 rz -54.03 deg; joints [-13.835, -58.533, 111.285, 192.985, 37.16, -113.331, -415]
  MoveL 5817 to (-41.03, 47.35, -221.61) mm, rotated rx -9.61 ry -16.54 rz -54.03 deg; joints [-13.835, -58.533, 111.285, 192.985, 37.16, -113.33, -415]
  MoveL 5818 to (-41.03, 47.9, -221.63) mm, rotated rx -9.61 ry -16.54 rz -54.03 deg; joints [-13.834, -58.496, 111.262, 192.982, 37.174, -113.326, -415]
  MoveL 5819 to (-41.01, 48.43, -221.68) mm, rotated rx -9.61 ry -16.54 rz -54.03 deg; joints [-13.834, -58.459, 111.241, 192.978, 37.188, -113.321, -415]
  MoveL 5820 to (-40.98, 49.01, -221.75) mm, rotated rx -9.61 ry -16.54 rz -54.03 deg; joints [-13.835, -58.42, 111.218, 192.971, 37.204, -113.314, -415]
  MoveL 5821 to (-40.97, 49.61, -221.79) mm, rotated rx -9.61 ry -16.54 rz -54.03 deg; joints [-13.834, -58.38, 111.194, 192.967, 37.22, -113.308, -415]
  MoveL 5822 to (-40.97, 50.82, -221.81) mm, rotated rx -9.61 ry -16.54 rz -54.03 deg; joints [-13.831, -58.298, 111.142, 192.964, 37.25, -113.3, -415]
  MoveL 5823 to (-40.96, 51.38, -221.84) mm, rotated rx -9.61 ry -16.54 rz -54.03 deg; joints [-13.83, -58.261, 111.12, 192.961, 37.265, -113.295, -415]
  MoveL 5824 to (-40.93, 51.85, -221.92) mm, rotated rx -9.61 ry -16.54 rz -54.03 deg; joints [-13.832, -58.229, 111.102, 192.954, 37.278, -113.289, -415]
  MoveL 5825 to (-40.88, 52.29, -222.01) mm, rotated rx -9.61 ry -16.54 rz -54.03 deg; joints [-13.834, -58.199, 111.086, 192.947, 37.291, -113.282, -415]
  MoveL 5826 to (-40.85, 52.71, -222.07) mm, rotated rx -9.61 ry -16.54 rz -54.03 deg; joints [-13.835, -58.171, 111.07, 192.941, 37.303, -113.276, -415]
  MoveL 5827 to (-40.84, 53.16, -222.1) mm, rotated rx -9.61 ry -16.54 rz -54.03 deg; joints [-13.835, -58.14, 111.051, 192.938, 37.315, -113.272, -415]
  MoveL 5828 to (-40.9, 55.78, -222.1) mm, rotated rx -9.61 ry -16.54 rz -54.03 deg; joints [-13.825, -57.963, 110.937, 192.935, 37.377, -113.258, -415]
  MoveL 5829 to (-40.69, 58.68, -222.45) mm, rotated rx -9.61 ry -16.54 rz -54.03 deg; joints [-13.83, -57.768, 110.826, 192.903, 37.459, -113.222, -415]
  MoveL 5830 to (-40.38, 59.92, -222.88) mm, rotated rx -9.61 ry -16.54 rz -54.03 deg; joints [-13.844, -57.685, 110.791, 192.866, 37.504, -113.191, -415]
  MoveL 5831 to (-39.93, 61.03, -223.48) mm, rotated rx -9.61 ry -16.54 rz -54.03 deg; joints [-13.867, -57.611, 110.77, 192.816, 37.553, -113.15, -415]
  MoveL 5832 to (-39.34, 62, -224.26) mm, rotated rx -9.61 ry -16.54 rz -54.03 deg; joints [-13.898, -57.546, 110.763, 192.751, 37.605, -113.099, -415]
  MoveL 5833 to (-38.61, 62.84, -225.21) mm, rotated rx -9.61 ry -16.54 rz -54.03 deg; joints [-13.936, -57.491, 110.77, 192.673, 37.66, -113.04, -415]
  MoveL 5834 to (-36.73, 64.09, -227.62) mm, rotated rx -9.61 ry -16.54 rz -54.03 deg; joints [-14.039, -57.408, 110.824, 192.475, 37.78, -112.894, -415]
  MoveL 5835 to (-34.88, 64.56, -230.04) mm, rotated rx -9.61 ry -16.54 rz -54.03 deg; joints [-14.144, -57.378, 110.909, 192.28, 37.88, -112.754, -415]
  MoveL 5836 to (-34.19, 64.4, -230.99) mm, rotated rx -9.61 ry -16.54 rz -54.03 deg; joints [-14.186, -57.388, 110.954, 192.205, 37.908, -112.702, -415]
  MoveL 5837 to (-33.65, 63.99, -231.76) mm, rotated rx -9.61 ry -16.54 rz -54.03 deg; joints [-14.222, -57.416, 111.001, 192.144, 37.923, -112.661, -415]
  MoveL 5838 to (-33.44, 63.68, -232.08) mm, rotated rx -9.61 ry -16.54 rz -54.03 deg; joints [-14.237, -57.436, 111.026, 192.119, 37.925, -112.645, -415]
  MoveL 5839 to (-33.27, 63.31, -232.36) mm, rotated rx -9.61 ry -16.54 rz -54.03 deg; joints [-14.251, -57.461, 111.05, 192.098, 37.923, -112.632, -415]
  MoveL 5840 to (-33.04, 62.38, -232.8) mm, rotated rx -9.61 ry -16.54 rz -54.03 deg; joints [-14.273, -57.523, 111.101, 192.067, 37.909, -112.615, -415]
  MoveL 5841 to (-32.97, 61.19, -233.05) mm, rotated rx -9.61 ry -16.54 rz -54.03 deg; joints [-14.289, -57.602, 111.153, 192.05, 37.881, -112.61, -415]
  MoveL 5842 to (-33.05, 59.74, -233.14) mm, rotated rx -9.61 ry -16.54 rz -54.03 deg; joints [-14.297, -57.698, 111.207, 192.048, 37.839, -112.616, -415]
  MoveL 5843 to (-33.1, 59.22, -233.14) mm, rotated rx -9.61 ry -16.54 rz -54.03 deg; joints [-14.299, -57.732, 111.225, 192.05, 37.823, -112.62, -415]
  MoveL 5844 to (-33.16, 58.77, -233.11) mm, rotated rx -9.61 ry -16.54 rz -54.03 deg; joints [-14.299, -57.762, 111.24, 192.054, 37.808, -112.625, -415]
  MoveL 5845 to (-33.24, 58.36, -233.05) mm, rotated rx -9.61 ry -16.54 rz -54.03 deg; joints [-14.298, -57.789, 111.252, 192.06, 37.793, -112.631, -415]
  MoveL 5846 to (-33.32, 57.96, -232.98) mm, rotated rx -9.61 ry -16.54 rz -54.03 deg; joints [-14.296, -57.816, 111.264, 192.067, 37.779, -112.638, -415]
  MoveL 5847 to (-33.4, 57.53, -232.94) mm, rotated rx -9.61 ry -16.54 rz -54.03 deg; joints [-14.295, -57.845, 111.277, 192.072, 37.764, -112.644, -415]
  MoveL 5848 to (-33.46, 57.02, -232.92) mm, rotated rx -9.61 ry -16.54 rz -54.03 deg; joints [-14.296, -57.878, 111.294, 192.075, 37.748, -112.649, -415]
  MoveL 5849 to (-34.03, 51.32, -232.91) mm, rotated rx -9.61 ry -16.54 rz -54.03 deg; joints [-14.314, -58.256, 111.49, 192.096, 37.567, -112.694, -415]
  MoveL 5850 to (-34.12, 50.56, -232.89) mm, rotated rx -9.61 ry -16.54 rz -54.03 deg; joints [-14.316, -58.307, 111.515, 192.1, 37.542, -112.701, -415]
  MoveL 5851 to (-34.23, 49.91, -232.89) mm, rotated rx -9.61 ry -16.54 rz -54.03 deg; joints [-14.318, -58.349, 111.534, 192.104, 37.519, -112.708, -415]
  MoveL 5852 to (-34.4, 49.37, -232.87) mm, rotated rx -9.61 ry -16.54 rz -54.03 deg; joints [-14.318, -58.384, 111.543, 192.111, 37.493, -112.716, -415]
  MoveL 5853 to (-34.64, 48.88, -232.83) mm, rotated rx -9.61 ry -16.54 rz -54.03 deg; joints [-14.317, -58.415, 111.546, 192.12, 37.467, -112.727, -415]
  MoveL 5854 to (-34.83, 48.61, -232.67) mm, rotated rx -9.61 ry -16.54 rz -54.03 deg; joints [-14.311, -58.432, 111.545, 192.135, 37.449, -112.739, -415]
  MoveL 5855 to (-34.85, 48.63, -232.36) mm, rotated rx -9.61 ry -16.54 rz -54.03 deg; joints [-14.298, -58.433, 111.547, 192.155, 37.452, -112.751, -415]
  MoveL 5856 to (-34.68, 48.95, -231.88) mm, rotated rx -9.61 ry -16.54 rz -54.03 deg; joints [-14.278, -58.417, 111.554, 192.179, 37.477, -112.762, -415]
  MoveL 5857 to (-35.3, 49.04, -230.91) mm, rotated rx -9.61 ry -16.54 rz -54.03 deg; joints [-14.235, -58.412, 111.517, 192.255, 37.452, -112.815, -415]
  MoveL 5858 to (-36.53, 47.63, -230.61) mm, rotated rx -9.61 ry -16.54 rz -54.03 deg; joints [-14.221, -58.496, 111.487, 192.309, 37.342, -112.868, -415]
  MoveL 5859 to (-37.8, 46.13, -230.4) mm, rotated rx -9.61 ry -16.54 rz -54.03 deg; joints [-14.211, -58.583, 111.455, 192.358, 37.226, -112.92, -415]
  MoveL 5860 to (-39.17, 44.5, -230.27) mm, rotated rx -9.61 ry -16.54 rz -54.03 deg; joints [-14.205, -58.678, 111.419, 192.405, 37.1, -112.973, -415]
  MoveL 5861 to (-41.88, 41.21, -230.27) mm, rotated rx -9.61 ry -16.54 rz -54.03 deg; joints [-14.202, -58.867, 111.346, 192.485, 36.844, -113.07, -415]
  MoveL 5862 to (-43.14, 39.68, -230.18) mm, rotated rx -9.61 ry -16.54 rz -54.03 deg; joints [-14.197, -58.956, 111.313, 192.528, 36.726, -113.119, -415]
  MoveL 5863 to (-44.5, 38.04, -230.18) mm, rotated rx -9.61 ry -16.54 rz -54.03 deg; joints [-14.195, -59.05, 111.276, 192.569, 36.598, -113.168, -415]
  MoveL 5864 to (-45.95, 36.43, -230.18) mm, rotated rx -9.61 ry -16.54 rz -54.03 deg; joints [-14.193, -59.139, 111.229, 192.613, 36.465, -113.22, -415]
  MoveL 5865 to (-47.68, 34.57, -230.01) mm, rotated rx -9.61 ry -16.54 rz -54.03 deg; joints [-14.183, -59.244, 111.173, 192.677, 36.31, -113.29, -415]
  MoveL 5866 to (-49, 32.78, -229.77) mm, rotated rx -9.61 ry -16.54 rz -54.03 deg; joints [-14.173, -59.349, 111.147, 192.732, 36.183, -113.349, -415]
  MoveL 5867 to (-50.3, 31.04, -229.65) mm, rotated rx -9.61 ry -16.54 rz -54.03 deg; joints [-14.167, -59.45, 111.118, 192.781, 36.057, -113.403, -415]
  MoveL 5868 to (-51.66, 29.39, -229.55) mm, rotated rx -9.61 ry -16.54 rz -54.03 deg; joints [-14.161, -59.544, 111.08, 192.83, 35.93, -113.459, -415]
  MoveL 5869 to (-53.01, 27.74, -229.33) mm, rotated rx -9.61 ry -16.54 rz -54.03 deg; joints [-14.151, -59.638, 111.044, 192.887, 35.804, -113.519, -415]
  MoveL 5870 to (-54.36, 26.09, -229.22) mm, rotated rx -9.61 ry -16.54 rz -54.03 deg; joints [-14.145, -59.731, 111.006, 192.937, 35.677, -113.575, -415]
  MoveL 5871 to (-55.71, 24.44, -229.11) mm, rotated rx -9.61 ry -16.54 rz -54.03 deg; joints [-14.139, -59.824, 110.968, 192.988, 35.55, -113.632, -415]
  MoveL 5872 to (-57.05, 22.78, -228.9) mm, rotated rx -9.61 ry -16.54 rz -54.03 deg; joints [-14.129, -59.919, 110.932, 193.045, 35.425, -113.693, -415]
  MoveL 5873 to (-58.4, 21.12, -228.8) mm, rotated rx -9.61 ry -16.54 rz -54.03 deg; joints [-14.124, -60.012, 110.894, 193.096, 35.298, -113.75, -415]
  MoveL 5874 to (-59.75, 19.47, -228.69) mm, rotated rx -9.61 ry -16.54 rz -54.03 deg; joints [-14.118, -60.104, 110.855, 193.148, 35.171, -113.808, -415]
  MoveL 5875 to (-61.07, 17.8, -228.48) mm, rotated rx -9.61 ry -16.54 rz -54.03 deg; joints [-14.109, -60.198, 110.819, 193.206, 35.045, -113.87, -415]
  MoveL 5876 to (-62.42, 16.14, -228.38) mm, rotated rx -9.61 ry -16.54 rz -54.03 deg; joints [-14.103, -60.291, 110.78, 193.258, 34.918, -113.928, -415]
  MoveL 5877 to (-63.52, 14.66, -228.12) mm, rotated rx -9.61 ry -16.54 rz -54.03 deg; joints [-14.092, -60.376, 110.755, 193.313, 34.812, -113.984, -415]
  MoveL 5878 to (-64.47, 13.28, -227.76) mm, rotated rx -9.61 ry -16.54 rz -54.03 deg; joints [-14.077, -60.456, 110.738, 193.37, 34.72, -114.04, -415]
  MoveL 5879 to (-65.28, 11.99, -227.26) mm, rotated rx -9.61 ry -16.54 rz -54.03 deg; joints [-14.057, -60.535, 110.732, 193.431, 34.641, -114.096, -415]
  MoveL 5880 to (-64.38, 12.68, -226.41) mm, rotated rx -9.61 ry -16.54 rz -54.03 deg; joints [-14.026, -60.509, 110.788, 193.456, 34.725, -114.097, -415]
  MoveL 5881 to (-64.59, 12.43, -226.38) mm, rotated rx -9.61 ry -16.54 rz -54.03 deg; joints [-14.024, -60.523, 110.782, 193.465, 34.706, -114.107, -415]
  MoveL 5882 to (-64.82, 12.2, -226.34) mm, rotated rx -9.61 ry -16.54 rz -54.03 deg; joints [-14.022, -60.535, 110.773, 193.476, 34.686, -114.118, -415]
  MoveL 5883 to (-65.14, 12.01, -226.29) mm, rotated rx -9.61 ry -16.54 rz -54.03 deg; joints [-14.019, -60.543, 110.757, 193.49, 34.662, -114.132, -415]
  MoveL 5884 to (-65.51, 11.83, -226.25) mm, rotated rx -9.61 ry -16.54 rz -54.03 deg; joints [-14.016, -60.55, 110.734, 193.505, 34.634, -114.147, -415]
  MoveL 5885 to (-65.97, 11.67, -226.22) mm, rotated rx -9.61 ry -16.54 rz -54.03 deg; joints [-14.013, -60.555, 110.705, 193.521, 34.602, -114.164, -415]
  MoveL 5886 to (-70.48, 10.31, -226.22) mm, rotated rx -9.61 ry -16.54 rz -54.03 deg; joints [-13.993, -60.577, 110.402, 193.667, 34.288, -114.322, -415]
  MoveL 5887 to (-70.86, 10.18, -226.2) mm, rotated rx -9.61 ry -16.54 rz -54.03 deg; joints [-13.99, -60.581, 110.378, 193.681, 34.262, -114.336, -415]
  MoveL 5888 to (-71.36, 10.03, -226.2) mm, rotated rx -9.61 ry -16.54 rz -54.03 deg; joints [-13.988, -60.583, 110.344, 193.697, 34.227, -114.354, -415]
  MoveL 5889 to (-72.34, 9.71, -226.16) mm, rotated rx -9.61 ry -16.54 rz -54.03 deg; joints [-13.982, -60.59, 110.28, 193.732, 34.159, -114.391, -415]
  MoveL 5890 to (-74.85, 8.96, -226.16) mm, rotated rx -9.61 ry -16.54 rz -54.03 deg; joints [-13.971, -60.601, 110.11, 193.815, 33.985, -114.48, -415]
  MoveL 5891 to (-75.82, 8.61, -226.14) mm, rotated rx -9.61 ry -16.54 rz -54.03 deg; joints [-13.966, -60.61, 110.047, 193.848, 33.916, -114.516, -415]
  MoveL 5892 to (-77.2, 8.17, -226.21) mm, rotated rx -9.61 ry -16.54 rz -54.03 deg; joints [-13.962, -60.616, 109.953, 193.89, 33.819, -114.563, -415]
  MoveL 5893 to (-78.35, 7.96, -226.46) mm, rotated rx -9.61 ry -16.54 rz -54.03 deg; joints [-13.967, -60.61, 109.866, 193.911, 33.74, -114.593, -415]
  MoveL 5894 to (-79.28, 7.97, -226.9) mm, rotated rx -9.61 ry -16.54 rz -54.03 deg; joints [-13.979, -60.591, 109.786, 193.912, 33.678, -114.605, -415]
  MoveL 5895 to (-79.66, 8.06, -227.19) mm, rotated rx -9.61 ry -16.54 rz -54.03 deg; joints [-13.988, -60.577, 109.748, 193.905, 33.654, -114.605, -415]
  MoveL 5896 to (-79.99, 8.2, -227.53) mm, rotated rx -9.61 ry -16.54 rz -54.03 deg; joints [-14, -60.56, 109.712, 193.893, 33.634, -114.6, -415]
  MoveL 5897 to (-80.46, 8.65, -228.34) mm, rotated rx -9.61 ry -16.54 rz -54.03 deg; joints [-14.028, -60.516, 109.645, 193.853, 33.608, -114.578, -415]
  MoveL 5898 to (-80.72, 9.33, -229.34) mm, rotated rx -9.61 ry -16.54 rz -54.03 deg; joints [-14.064, -60.459, 109.585, 193.792, 33.599, -114.538, -415]
  MoveL 5899 to (-80.55, 11.33, -231.89) mm, rotated rx -9.61 ry -16.54 rz -54.03 deg; joints [-14.159, -60.308, 109.485, 193.611, 33.633, -114.407, -415]
  MoveL 5900 to (-79.61, 13.54, -234.46) mm, rotated rx -9.61 ry -16.54 rz -54.03 deg; joints [-14.258, -60.155, 109.436, 193.404, 33.72, -114.249, -415]
  MoveL 5901 to (-78.05, 15.28, -236.29) mm, rotated rx -9.61 ry -16.54 rz -54.03 deg; joints [-14.334, -60.049, 109.466, 193.229, 33.84, -114.107, -415]
  MoveL 5902 to (-77.03, 15.97, -236.93) mm, rotated rx -9.61 ry -16.54 rz -54.03 deg; joints [-14.362, -60.014, 109.51, 193.153, 33.913, -114.042, -415]
  MoveL 5903 to (-75.86, 16.54, -237.39) mm, rotated rx -9.61 ry -16.54 rz -54.03 deg; joints [-14.385, -59.99, 109.574, 193.085, 33.995, -113.981, -415]
  MoveL 5904 to (-73.05, 17.32, -237.76) mm, rotated rx -9.61 ry -16.54 rz -54.03 deg; joints [-14.413, -59.978, 109.76, 192.972, 34.185, -113.87, -415]
